		(* Check input high *)
		ELSIF
			BitInToCheck AND
			InputAvailable AND
			NOT CheckSignalLow AND
			CheckSignalHigh THEN

			TimerTimeOut(Start := FALSE, MTime := (sInit.MaxTime));
			State:=State_OK;
	
		(* Check signal high and input is low*)
		ELSIF
			NOT BitInToCheck AND
			InputAvailable AND
			NOT CheckSignalLow AND
			CheckSignalHigh THEN

			TimerTimeOut(Start := TRUE, MTime := (sInit.MaxTime));
			State:=STATE_ERROR (*INPUT_CHECKHIGH*);
			FB_ReadXmlLineMsg.ID:='SensorFaultNotHigh';

			TempErrorText:=sVisu.InstName;
			TempErrorText:=CONCAT(TempErrorText,' :');
			TempErrorText:=CONCAT(TempErrorText,sVisu.Description);
			TempErrorText:=CONCAT(TempErrorText,'  ');
			TempErrorText:=CONCAT(TempErrorText,FB_ReadXmlLineMsg.Text);

			Error.No:=2;
		ELSE
			TimerTimeOut(Start := FALSE, MTime := (sInit.MaxTime));

			IF	SetSignalHigh AND
				CheckSignalLow AND
				NOT PulseOn AND
				NOT FlashSignal AND
				NOT CheckSignalHigh AND
				NOT CheckSignalLow THEN

				State:=STATE_WAIT;
			END_IF
		END_IF

		(* Timeout check high *)
		IF	TimerTimeOut.Timeout AND
			NOT ResetIntern AND
			State=INPUT_CHECKHIGH 	THEN

			State:=STATE_ERROR (*INPUT_CHECKHIGHFAULT*);
			FB_ReadXmlLineMsg.ID:='NotHhigh';

			TempErrorText:=sVisu.InstName;
			TempErrorText:=CONCAT(TempErrorText,' ');
			TempErrorText:=CONCAT(TempErrorText,sVisu.Description);
			TempErrorText:=CONCAT(TempErrorText,' ');
			TempErrorText:=CONCAT(TempErrorText,FB_ReadXmlLineMsg.Text);
			Error.No:=3;
		END_IF
		(* Timeout check low *)
		IF	TimerTimeOut.Timeout AND
			NOT ResetIntern AND
			State=INPUT_CHECKLOW THEN

			State:=STATE_ERROR (*INPUT_CHECKLOWFAULT*);
			FB_ReadXmlLineMsg.ID:='NotLow';

			TempErrorText:=sVisu.InstName;
			TempErrorText:=CONCAT(TempErrorText,' ');
			TempErrorText:=CONCAT(TempErrorText,sVisu.Description);
			TempErrorText:=CONCAT(TempErrorText,' ');
			TempErrorText:=CONCAT(TempErrorText,FB_ReadXmlLineMsg.Text);
			Error.No:=4;
		END_IF

	ELSE	(* No action *)
		(* Reset ok signal*)
		IF 	State = State_OK AND
			StateOK_CycleFlag THEN

			State:=STATE_WAIT;
		END_IF
	END_IF

END_IF	(* Init ok *)

(*--------------------------------------------------------------------
	Updating processtime (if State_RUN, STATE_ERROR, STATE_RESETS, or STATE_STOPPED)
--------------------------------------------------------------------*)
IF	( State=State_RUN OR
	State=STATE_ERROR OR
	State=STATE_RESETS OR
	State=STATE_STOPPED ) AND
	sInit.MaxTime<>0 AND
	InputAvailable<>0 THEN

	TimerTimeOut;
	ProcessTime:=TimerTimeOut.PTime;
END_IF

(*------------------------------------------------------------------
	Reset-Handling
  ------------------------------------------------------------------*)
ResetIntern:=Reset;

IF 	ResetIntern THEN

	TimerTimeOut (Start := FALSE, MTime := (sInit.MaxTime));
	State:= STATE_RESETS;
	BitOutToSet:=FALSE;
	SetOutPulse(IN:=FALSE);
	TimerOn(IN:=FALSE);
	TimerOff(IN:=FALSE);

	SetSignalHigh:=FALSE;		 		 	(* Signal set  HIGH *)
	SetSignalLow:=FALSE;		 			(* Signal set  LOW  *)
	PulseOn:=FALSE;		 			(* Signal pulse On *)
	FlashSignal:=FALSE;		 			(* Signal FLASH  *)
ELSE  (* IF Reset=FALSE *)
	IF 	State=STATE_RESETS THEN
		State:=STATE_WAIT;
	END_IF
END_IF

(*------------------------------------------------------------------
	Clear all input variables
  ------------------------------------------------------------------*)
Reset:= FALSE;
SetSignalLow:=FALSE;
SetSignalHigh:=FALSE;
PulseOn:=FALSE;
FlashSignal:=FALSE;
CheckSignalLow:= FALSE;
CheckSignalHigh:= FALSE;

(*------------------------------------------------------------------
	HomePosition
  ------------------------------------------------------------------*)
HomePositionInfo:=State_OK;

(* Check input signal *)
IF	sInit.HomePosSignal=0 AND
	BitInToCheck AND
	InputAvailable THEN
	HomePositionInfo:=11;
END_IF

IF	sInit.HomePosSignal=1 AND
	NOT BitInToCheck AND
	InputAvailable THEN
	HomePositionInfo:=10;
END_IF

(* Check output signal *)
IF	sInit.HomePosOutput=0 AND
	BitOutToSet AND
	OutputAvailable THEN
	HomePositionInfo:=21;
END_IF

IF	sInit.HomePosOutput=1 AND
	NOT BitOutToSet AND
	OutputAvailable THEN
	HomePositionInfo:=20;
END_IF


(* Generating home position*)
(* Zuweisung der Grundstellung*)
IF HomePositionInfo=State_OK THEN
	HomePosition:= TRUE;
ELSE
	HomePosition:= FALSE;
	ListHomeNOK(InstName:=sInit.InstName,Description:=FB_ReadXmlLineConf.Text);
END_IF

(* Objekt-Grundstellung verknüpfen mit GesamtGrundstellung *)
(* object-homeposition concat with mainhomeposition *)
gHomeOk:=gHomeOk AND HomePosition;

(*------------------------------------------------------------------
	Set Visu-Vars
  ------------------------------------------------------------------*)
sVisu.BitInName			:= sInit.BitInName;
sVisu.BitOutToSet		:= BitOutToSet;
sVisu.BitInToCheck		:= BitInToCheck;
sVisu.State				:= State;
sVisu.HomePosition		:= HomePosition;


(*Copy output-signal to output-var*)
SignalOut:=BitOutToSet;
(*Copy input-signal to output-var*)
SignalIn:=BitInToCheck;

(*------------------------------------------------------------------
	Error-Handling
  ------------------------------------------------------------------*)
ErrorElapsed(CLK:= Error.Text<>'');
IF ErrorElapsed.Q THEN
	Error.DateTime:=gVarDTSystemtime;
END_IF

IF Error.Text<>''	AND ST_Lng.b_EndChangeLng THEN
	Error.Typ:=0;

	(*Error.DateTime:=;*)
	ErrorHandler.AddError(
			ErrorToAdd:=Error,
			sVisu:=Visu.ErrorHandler);
END_IF

IF 	NOT Enable AND ModeSelect.Mode=MODE_MANUAL AND
	Error.Text='' AND
	strAnlayse<>'' THEN

	strAnlayse:=CONCAT(' +++ gesperrt durch : ',strAnlayse);

	LaufschriftAnalyse(
	N:= 40,
	StepWidth:=1,
	PT:= t#100ms ,
	Text:= strAnlayse,
	Display=>sVisu.ErrorString );

	strAnlayse:='';
ELSE
	IF Error.Text<>''	THEN
		TempString:=CONCAT(' --- ',Error.Text);
		LaufschriftObj(
		N:= 40,
		StepWidth:=1,
		PT:= t#100ms ,
		Text:= TempString,
		Display=>sVisu.ErrorString );
	ELSE
		sVisu.ErrorString:='';
	END_IF
END_IF

sVisu.InstName:=sInit.InstName;
sVisu.BitOutName:=sInit.BitOutName;
sVisu.BitInName:=sInit.BitInName;
sVisu.ErrorPresent:=Error.Text<>'';

FB_ReadXmlLineConf(
	Prefix:= 'CONFIG',
	ID:= sInit.InstName,
	File:= 'CONFIG.xml',
	Text=> sVisu.Description);

FB_ReadXmlLineMsg(
	Prefix:= 'MSG',
	ID:= ,
	File:= 'MSG.xml',
	Text=>);

IF 	State = STATE_ERROR THEN
	TempErrorText:=sInit.BitInName;
	TempErrorText:=CONCAT(TempErrorText,' :');
	TempErrorText:=CONCAT(TempErrorText,sVisu.Description);
	TempErrorText:=CONCAT(TempErrorText,' -> ');
	TempErrorText:=CONCAT(TempErrorText,FB_ReadXmlLineMsg.Text);
END_IF
END_FUNCTION_BLOCK

(* POU zLibrary/AnaIn/FB_Encoder, ST *)
FUNCTION_BLOCK FB_Encoder
VAR_INPUT
	sInit					:sEncoderInit;	(* Initializingvalues to the Instance *)
	Reset					:BOOL;
END_VAR
VAR_OUTPUT
	State					:StateObject;	(* State of the object *)
	rpmValue			: LREAL;		(* rpm *)
	posValue			: LREAL;		(* mm *)
	Drehrichtung		: enum_Drehrichtung;
END_VAR
VAR_IN_OUT
	sVisu				:sEncoderVisu;
END_VAR
VAR

	Error					:ErrorStruct;
	TempErrorText			:STRING(255);
	ErrorElapsed			:BOOL;
	LaufschriftErrh			:FB_Laufschrift;
	LaufschriftObj			:FB_Laufschrift_STR255;
	InitState				:BOOL:=FALSE;	(* Internal State for initialising *)



	FB_ReadXmlLineConf		:FB_ReadXmlLine;
	FB_ReadXmlLineMsg		:FB_ReadXmlLine;
END_VAR


(*==================================================================*)
VAR_OUTPUT

END_VAR

VAR
	fb_ton_Reset		: TON;
	fb_ton_steht		: TON;
	fb_ton_dreht		: TON;

	fb_rTrigReset		: R_TRIG;
	fb_rTrigUnderflow		: R_TRIG;
	fb_rTrigOverflow		: R_TRIG;

	i_count_ueberlauf		: DINT;		(* +- 64bit *)
	lr_xBit		: LREAL;
	lr_rpmHelp	: LREAL;	(*°*)

	
	e_Value					AT %I* : UINT;		(* 65535 *)
	e_CountUnderflow		AT %I* : BOOL;
	e_CountOverflow			AT %I* : BOOL;
	a_CountReset			AT %Q* : BOOL;

END_VAR
VAR CONSTANT



END_VAR
Error.No:=0;
Error.Text:='';

(*------------------------------------------------------------------
	Initialization
  ------------------------------------------------------------------*)
IF  NOT InitState THEN
	InitState:=TRUE;
	State:=STATE_OK;
	(* Check instance name *)
	IF 	sInit.InstName=''THEN
		InitState:=FALSE;
		State:=STATE_ERROR;
		FB_ReadXmlLineMsg.ID:='InstNameNotDefined';

		TempErrorText:=sInit.BitInName;
		TempErrorText:=CONCAT(TempErrorText,' :');
		TempErrorText:=CONCAT(TempErrorText,sVisu.Description);
  		TempErrorText:=CONCAT(TempErrorText,' -> ');
		TempErrorText:=CONCAT(TempErrorText,FB_ReadXmlLineMsg.Text);
		Error.No:=4;
	(*CheckDescription*)
	ELSIF
		sInit.Description=''THEN
		InitState:=FALSE;
		State:=STATE_ERROR;
		FB_ReadXmlLineMsg.ID:='DescriptionNotDefined';

		TempErrorText:=sInit.BitInName;
		TempErrorText:=CONCAT(TempErrorText,' :');
		TempErrorText:=CONCAT(TempErrorText,sVisu.Description);
  		TempErrorText:=CONCAT(TempErrorText,' -> ');
		TempErrorText:=CONCAT(TempErrorText,FB_ReadXmlLineMsg.Text);
		Error.No:=4;
	ELSIF
		sInit.i_InkProRpm=0THEN
		InitState:=FALSE;
		State:=STATE_ERROR;
		FB_ReadXmlLineMsg.ID:='InkProRpmNotDefined';

		TempErrorText:=sInit.BitInName;
		TempErrorText:=CONCAT(TempErrorText,' :');
		TempErrorText:=CONCAT(TempErrorText,sVisu.Description);
  		TempErrorText:=CONCAT(TempErrorText,' -> ');
		TempErrorText:=CONCAT(TempErrorText,FB_ReadXmlLineMsg.Text);
		Error.No:=4;
	END_IF

END_IF

(* Add InitState to Global-Init-State to collect all Objects *)
gInitCollect:=gInitCollect AND InitState;

(*==================================================================*)
IF  InitState THEN
	(* Drehrichtung ermitteln *)
	fb_ton_steht(PT:=T#50MS);
	IF	lr_rpmHelp > rpmValue - 0.0001 AND
		lr_rpmHelp < rpmValue + 0.0001 THEN
		fb_ton_steht.IN:=TRUE;
		IF	fb_ton_steht.Q THEN
			Drehrichtung:= STEHT;
		END_IF
	ELSIF
		lr_rpmHelp < rpmValue THEN
		fb_ton_steht.IN:=FALSE;
		Drehrichtung:= VORWAERTS;
	ELSIF
		lr_rpmHelp > rpmValue THEN
		fb_ton_steht.IN:=FALSE;
		Drehrichtung:= RUECKWAERTS;
	END_IF
	lr_rpmHelp:=rpmValue;
	
	(* Encoderüberlauf*)
	fb_rTrigUnderflow(CLK:= e_CountUnderflow);
	fb_rTrigOverflow(CLK:= e_CountOverflow);
	IF 	fb_rTrigUnderflow.Q THEN
		i_count_ueberlauf:=i_count_ueberlauf - 1;
	ELSIF
		fb_rTrigOverflow.Q THEN
		i_count_ueberlauf:=i_count_ueberlauf + 1;
	END_IF

	(* bei Reset Nullen *)
	fb_ton_Reset(IN:=Reset , PT:= T#300MS , Q=> , ET=> );
	a_CountReset:=Reset OR sVisu.Reset;
	fb_rTrigReset(CLK:=fb_ton_Reset.Q, );
	IF	fb_rTrigReset.Q THEN
		Reset:=FALSE;
	END_IF

	(* aktuelle Position *)
	IF	e_Value <> 0 THEN
		lr_xBit:=EXPT(2,16);												(* 16 bit=65535  Inkremente Encoder*)
		rpmValue:= e_Value + (lr_xBit * DINT_TO_LREAL(i_count_ueberlauf));	(* Inkremente*)
		rpmValue:= rpmValue / sInit.i_InkProRpm;							(* Umdrehungen in Grad*)
	ELSE
		rpmValue:= 0;
		i_count_ueberlauf:=0;
	END_IF
	IF	sInit.lr_LaengeProRpm > 0 THEN
		posValue:= rpmValue * sInit.lr_LaengeProRpm;					(* Strecke in mm*)
	ELSE
		posValue:= 0;													(* Strecke in mm*)
	END_IF

	sVisu.posValue:=posValue;
	sVisu.rpmValue:=rpmValue;
	sVisu.Drehrichtung:=Drehrichtung;
END_IF
(* ------------------------------------------------------------------------------------------ *)
(* ---------------- LANGUAGE auslesen aus der XML Datei-------- *)
(* ------------------------------------------------------------------------------------------ *)
sVisu.BitInName:=sInit.BitInName;
sVisu.InstName:=sInit.InstName;
sVisu.ErrorPresent:=Error.Text<>'';

(*  *)
IF 	State=STATE_ERROR AND
	NOT ErrorElapsed THEN
	ErrorElapsed:=TRUE;
	Error.DateTime:=gVarDTSystemtime;
ELSIF
	State<>STATE_ERROR THEN
	ErrorElapsed:=FALSE;
	TempErrorText:='';
END_IF;

IF 	Error.Text<>'' AND
	ST_Lng.b_EndChangeLng THEN
	(*Error.DateTime:=;*)
	Error.Typ:=0;
	ErrorHandler.AddError(ErrorToAdd:=Error,
	sVisu:=Visu.ErrorHandler);
END_IF


FB_ReadXmlLineConf(
	Prefix:= 'CONFIG',
	ID:= sInit.InstName,
	File:= 'CONFIG.xml',
	Text=> sVisu.Description  );

FB_ReadXmlLineMsg(
	Prefix:= 'MSG',
	ID:= ,
	File:= 'MSG.xml',
	Text=>);

IF 	State = STATE_ERROR THEN
	TempErrorText:=sInit.BitInName;
	TempErrorText:=CONCAT(TempErrorText,' :');
	TempErrorText:=CONCAT(TempErrorText,sVisu.Description);
	TempErrorText:=CONCAT(TempErrorText,' -> ');
	TempErrorText:=CONCAT(TempErrorText,FB_ReadXmlLineMsg.Text);
END_IF


LaufschriftErrh(
N:= 160,
StepWidth:=1,
PT:= t#100ms ,
Text:= TempErrorText,
Display=>Error.Text );

LaufschriftObj(
N:= 40,
StepWidth:=1,
PT:= t#100ms ,
Text:= TempErrorText,
Display=>sVisu.ErrorString );
END_FUNCTION_BLOCK

(* POU zLibrary/EpsonRobot/FB_EpsonRobot, ST *)
FUNCTION_BLOCK FB_EpsonRobot (*25.NOV 2010, Bernd Happach*)
VAR_INPUT
	ExecuteMove					: BOOL; 				(* Move to PositionNo *)
	PosNo							: DINT;					(* Position No from Robot *)
	PosOffset						: DINT;					(* Offset *)
	Override						: DINT;					(* Global override *)
	OffsetX							: REAL;					(* Offset X *)
	OffsetY							: REAL;					(* Offset Y *)
	OffsetZ							: REAL;					(* Offset Z *)
	ApplPara						: ARRAY[0..7] OF	REAL; (* Machinespecific Values *)

	SetToolOn						: BOOL;
	SetToolOff						: BOOL;

	Vel								: DINT;					(* Velocity for Linear Movements *)
	Acc								: DINT;					(* Acceleration 0..100% *)

	Enable							: BOOL; 				(* Enables the operations on the valve *)
	Reset							: BOOL; 				(* switch for resetting the object *)
	SFCCurrentStep					: STRING(80);			(* aktually step in the step flow chart *)
	SFCCurrentPOU					: STRING(80);			(* Name of the step flow chart *)
	sInit								: sEpsonRobotInit;		(* Initializingvalues to the Instance *)
	sToolSettings					: sEpsonRobotToolSettings;
	strAnlayse						: STRING(255);  		(*String to analyse Lockings*)

	CollisionActivated			:BOOL;
	Tool2Unit_AST						:BOOL;
END_VAR
VAR_OUTPUT
	State							: StateObject;			(* State of the object *)
	HomePosition					: BOOL;					(* object in home-position*)
	ActualPosition					: DINT;
	ActualArea						: DINT;
END_VAR
VAR_IN_OUT
	sVisu							: sEpsonRobotVisu;   	(* Structure for Visualisation *)
END_VAR
VAR
	RemOutStart					AT %Q* :	BOOL; 		(* Startbit für Task Main *)
	RemOutStop					AT %Q* :	BOOL; 		(* Task stoppen/ beenden *)
	RemOutPause					AT %Q* :	BOOL; 		(* Task anhalten *)
	RemOutCont					AT %Q* :	BOOL; 		(* Task fortsetzen *)
	RemOutReset					AT %Q* :	BOOL; 		(* Reset auf Roboter *)
	RemOutPowerOn				AT %Q* :	BOOL; 		(* Armleistung ein *)
	RemOutPowerOff				AT %Q* :	BOOL; 		(* Armleistung aus *)
	RemOutPowerHi					AT %Q* :	BOOL; 		(* Motor hohe Leistung ein *)
	RemOutSetToolOn				AT %Q* :	BOOL; 		(* Anforderung Ausgang Robotertool EIN *)
	RemOutSetToolOff				AT %Q* :	BOOL; 		(* Anforderung Ausgang Robotertool AUS *)

	RemInReady					AT %I* :	BOOL; 		(* Betriebsbereit von Roboter *)
	RemInRunning					AT %I* :	BOOL; 		(* Task (Main) aktiv von Roboter *)
	RemInPaused					AT %I* :	BOOL; 		(* Task angehalten - nicht abgebrochen! *)
	RemInError						AT %I* :	BOOL; 		(* quittierbare Störung von Roboter *)
	RemInEStopOn					AT %I* :	BOOL; 		(* Notaus-Kreis aktiv von Roboter *)
	RemInSafeguardOn				AT %I* :	BOOL; 		(* Schutzkreis (Türen) aktiv von Roboter *)
	RemInSError					AT %I* :	BOOL; 		(* nicht quittierbare Störung - Roboter AEG notwendig *)
	RemInWarning					AT %I* :	BOOL; 		(* Warnmeldung von Roboter *)
	RemInTcpIP_Wait				AT %I* :	BOOL; 		(* Handshake TcpIp-Verbindung *)
	RemInAreaBit1					AT %I* :	BOOL; 		(* Bereichsüberwachung Bit 1 *)
	RemInAreaBit2					AT %I* :	BOOL; 		(* Bereichsüberwachung Bit 2 *)
	RemInAreaBit4					AT %I* :	BOOL; 		(* Bereichsüberwachung Bit 4 *)

	RemInToolCoilA					AT %I* :  BOOL;		(* Rückmeldung Tool CoilA/ Ausgang 1 ist ein *)
	RemInToolCoilB					AT %I* :  BOOL;		(* Rückmeldung Tool CoilB/ Ausgang 2 ist ein *)
	RemInToolInitSensor				AT %I* :  BOOL;		(* Tool Ruhesensor *)
	RemInToolWorkSensor			AT %I* :  BOOL;		(* Tool Ruhesensor *)

	CollisionSensor					AT %I* :  BOOL;		(* Kollisonssensor Greifer*)

(* Internal used variables for movement Handling *)
	WorkingStep				: DINT;					(* Index for StateMachine *)
	PosNoLastMove				: DINT;					(* Position No from Robot *)
(* Init Handling *)
	InitStep						: INT;					(* Init Step StateMachine *)
	InitState						: BOOL :=	FALSE;		(* Internal State for initialising *)
	InitTimeOut					: TON;

	StepTimeOut				: TON;
(* Tool Handling *)
	ManToolOn					: TP;
	ManToolOff					: TP;

(* Error Handling *)
	TP_RemOutReset			: TP;

	TimerTimeOut				: CheckProcTime;	(* Timer generates timeout signal *)
	ProcessTime				: DINT;				(* Counts the time since starting operation *)

	Error						: ErrorStruct;
	ErrorElapsed				: R_TRIG;

	LaufschriftErrh				:FB_Laufschrift_STR255;
	LaufschriftObj				:FB_Laufschrift_STR255;
	LaufschriftAnalyse			:FB_Laufschrift_STR255;
	TempString					:STRING(255);

(* Internal used Variables tp send/receife data over TcpIP Socket *)
	ConnectionAlive				: BOOL;
	ConnectionTimer			: TON;
	TcpIP_Wait					: TON;
	ToolTimeOut				: TON;

	FP_Connected				: R_TRIG;


	DataIn						: sEpsonRobotRecvData;
	DataOut					: sEpsonRobotSendData;
	DataOutOld					: sEpsonRobotSendData;
	SendString					: STRING(255);

	ReceiveStep				: INT;

	FBClientServerConnection	: FB_ClientServerConnection;
	FBSocketReceive			: FB_SocketReceive;
	FBSocketSend				: FB_SocketSend;
	SocketHandle				: T_HSOCKET;

	_TON_SEND				: TP;

	eSocketState 				: E_SocketConnectionState;
	rxBuffer						: STRING(255);
	recString					: STRING(255);
	recBytes					: UDINT;

	StringWork					: STRING(255);
	ItemNo						: INT;
	StringStart					: INT;
	StringEnd					: INT;
	StringLen					: INT;
	ItemString					: STRING(255);
	ItemStringArray				: ARRAY [1..20] OF STRING;
	iPosArray					: INT;
(* Constants *)
	Delim						: STRING	:= ',';
	NoOfItems					: INT 		:= 16;


(* Visu Handling *)
	BtnMove					: VisuButton;
	BtnReset					: VisuButton;
	BtnPrgStart					: VisuButton;
	BtnPrgStop					: VisuButton;

	BtnToolOn					: VisuButton;
	BtnToolOff					: VisuButton;


	FB_ReadXmlLineConf		: FB_ReadXmlLine;
	FB_ReadXmlLineMsg		: FB_ReadXmlLine;

(*Kollisionsüberwachung*)
	fb_ton_collision				:TON;
	b_collision							: BOOL;
END_VAR
VAR CONSTANT
	RecBufferLen				: DINT := 100;
END_VAR
ToolTimeOut(IN:=,PT:=DINT_TO_TIME(sInit.ToolMaxTime));
Error.No:=0;
Error.Text:='';

Collision();
(*------------------------------------------------------------------
	Initialization
  ------------------------------------------------------------------*)
InitTimeOut(In:=NOT InitState,Pt:=T#5s);
IF 	NOT InitState THEN
	CASE InitStep OF
		0: (* Init Instance *)
			InitStep:=10;

		10:	InitStep:=50;
	
		50: (*Check IP-adress and Port*)
			InitStep:=100;

		100: (* Init Done *)
			IF	sInit.InstName <> '' THEN

				FOR iPosArray:=1 TO 20 DO
					(*Übersetzungen stehen in der CONFIG.xml*)
					sVisu.PosArray[iPosArray]:= '';
					sVisu.PosArray[iPosArray]:= CONCAT(	sVisu.PosArray[iPosArray],	sInit.InstName);
					sVisu.PosArray[iPosArray]:= CONCAT(	sVisu.PosArray[iPosArray],	'.PosArray[');
					sVisu.PosArray[iPosArray]:= CONCAT(	sVisu.PosArray[iPosArray],	INT_TO_STRING(iPosArray));
					sVisu.PosArray[iPosArray]:= CONCAT(	sVisu.PosArray[iPosArray],	']');
				END_FOR

			InitState:=TRUE;
			END_IF
	END_CASE

END_IF

IF InitState THEN
(*------------------------------------------------------------------
	Show and Read Visu Buttons
  ------------------------------------------------------------------*)
	BtnMove(	Button:=sVisu.BtnMove,
				Enable:=ModeSelect.Mode =	MODE_MANUAL AND
											Enable AND
											State=STATE_WAIT,
				TextOn:='Start'
							);

	BtnReset(	Button:=sVisu.BtnReset,
				Enable:=ModeSelect.Mode=MODE_MANUAL OR State=STATE_ERROR,
				TextOn:='Reset',
							);
	BtnPrgStart(	Button:=sVisu.BtnPrgStart,
				Enable:=ModeSelect.Mode=MODE_MANUAL ,
				TextOn:='Verbinden',
							);
	BtnPrgStop(	Button:=sVisu.BtnPrgStop,
				Enable:=ModeSelect.Mode=MODE_MANUAL ,
				TextOn:='Trennen',
							);
	BtnToolOn(	Button:=sVisu.BtnToolOn,
				Enable:=ModeSelect.Mode=MODE_MANUAL AND RemInRunning AND State=STATE_WAIT,
				TextOn:=sToolSettings.NameBtnToolOn,
							);
	BtnToolOff(	Button:=sVisu.BtnToolOff,
				Enable:=ModeSelect.Mode=MODE_MANUAL AND RemInRunning AND State=STATE_WAIT,
				TextOn:=sToolSettings.NameBtnToolOff,
							);
(*------------------------------------------------------------------
	EA-Handling
  ------------------------------------------------------------------*)
	ActualArea.0:=RemInAreaBit1;
	ActualArea.1:=RemInAreaBit2;
	ActualArea.2:=RemInAreaBit4;

	sVisu.ActualArea:=ActualArea;
(*------------------------------------------------------------------
	Manual Mode
  ------------------------------------------------------------------*)
	IF 	ModeSelect.Mode=MODE_MANUAL AND
		Enable THEN
		ExecuteMove:= BtnMove.Pressed;
		Reset:=Reset OR BtnReset.Pressed;
		IF 	ExecuteMove THEN
			(*Override:=10;*)
			PosNo:=sVisu.PosNo;
			OffsetX:=sVisu.OffsetX;
			OffsetY:=sVisu.OffsetY;
			OffsetZ:=sVisu.OffsetZ;
		END_IF

		ManToolOn(In:=BtnToolOn.Pressed,Pt:=T#1s);
		ManToolOff(In:=BtnToolOff.Pressed,Pt:=T#1s);
	END_IF

	RemOutPowerHi:=ModeSelect.Mode>MODE_MANUAL;
(*------------------------------------------------------------------
	Move-Handling
  ------------------------------------------------------------------*)
	TP_RemOutReset(In:=Reset,PT:=T#1s);

	RemOutReset:=	TP_RemOutReset.Q AND
					(	(	RemInError AND ( DataIn.ErrorCode < 8000 OR DataIn.ErrorCode > 8999 )	) OR
						RemInEStopOn OR
						RemInWarning OR
						RemInSError OR
						RemInSafeguardOn OR
						RemInPaused
						);
	RemOutPowerOff:=TP_RemOutReset.Q;
	RemOutCont:=TP_RemOutReset.Q;

	RemOutStart := 	(RemInReady AND
					NOT RemInRunning AND
					NOT RemInError AND
					NOT RemInEStopOn AND
					NOT RemInSafeguardOn AND
					NOT RemInSError AND
					NOT RemInWarning AND
					NOT TP_RemOutReset.Q AND
					vGlbImpuls_0500ms AND
					ModeSelect.Mode>MODE_MANUAL
					)	OR
					(RemInReady AND
					NOT RemInRunning AND
					NOT RemInError AND
					NOT RemInEStopOn AND
					NOT RemInSafeguardOn AND
					NOT RemInSError AND
					NOT RemInWarning AND
					NOT TP_RemOutReset.Q AND
					ModeSelect.Mode=MODE_MANUAL AND
					BtnPrgStart.Pressed
					);

	RemOutStop:= 	RemInRunning AND
					ModeSelect.Mode=MODE_MANUAL AND
					(BtnPrgStop.Pressed OR TP_RemOutReset.Q) OR
					RemInRunning AND
					ModeSelect.Mode>MODE_MANUAL AND
					TP_RemOutReset.Q;

	RemOutSetToolOn:=	(    ManToolOn.Q AND ModeSelect.Mode=MODE_MANUAL ) OR
						(    SetToolOn  AND ModeSelect.Mode>MODE_MANUAL );

	RemOutSetToolOff:=	 (  ManToolOff.Q AND ModeSelect.Mode=MODE_MANUAL ) OR
						 (  SetToolOff AND ModeSelect.Mode>MODE_MANUAL );

(* Generate Flags To Start Movement *)

	CASE WorkingStep OF
	0: (* State STATE_WAIT *)

		State:=STATE_WAIT;

		IF 	ExecuteMove THEN
			WorkingStep:=10;
			(* Start Execution Time *)
			TimerTimeOut.Start:=TRUE;
			State:=STATE_RUN;
		END_IF
	10: (* Check Star Conditions *)
		IF  ConnectionAlive AND
			RemInRunning THEN
			WorkingStep:=100;
		ELSE
			State:=STATE_ERROR;
		END_IF
	100:(* Handle Robot EA´s if nessecary *)
			StepTimeOut(In:=FALSE);
			WorkingStep:=200;
	200:(* Start Movement - Assign Variables *)

			PosNoLastMove:=PosNo + PosOffset;

			DataOut.TelNo:=2;
			DataOut.PosNo:=PosNo + PosOffset;
			DataOut.Override:=Override;
			DataOut.OffsetX:=OffsetX;
			DataOut.OffsetY:=OffsetY;
			DataOut.OffsetZ:=OffsetZ;
			DataOut.ApplPara:=ApplPara;
			DataOut.Vel:=Vel;
			DataOut.Acc:=Acc;

			StepTimeOut(In:=DataIn.TelNo<>0 AND DataIn.TelNo<>DataOut.TelNo,Pt:=DINT_TO_TIME(sInit.MaxTime));
			IF 	DataIn.TelNo=DataOut.TelNo THEN
				WorkingStep:=201;
				ActualPosition:=0;

			ELSIF StepTimeOut.Q THEN
				(* Error *)
				State:=STATE_ERROR;
				FB_ReadXmlLineMsg.ID:='StartError';
				Error.No:=1;
				Error.Text:=sInit.InstName;
				Error.Text:=CONCAT(Error.Text,': ');
				Error.Text:=CONCAT(Error.Text,sInit.Description);
				Error.Text:=CONCAT(Error.Text,' - ');
				Error.Text:=CONCAT(Error.Text,FB_ReadXmlLineMsg.Text);
				WorkingStep:=999;
			END_IF

	201:(* Dummy step *)
			StepTimeOut(In:=FALSE);
			WorkingStep:=210;

	210:(* Wait Movement Done *)
			StepTimeOut(In:=DataIn.PosNo <>0 AND DataIn.PosNo<>DataOut.PosNo,Pt:=DINT_TO_TIME(sInit.MaxTime));
			IF 	DataIn.PosNo=DataOut.PosNo THEN
				DataOut.TelNo:=0;
				DataOut.PosNo:=0;
				ActualPosition:=DataIn.PosNo;
				WorkingStep:=220;
			ELSIF
				StepTimeOut.Q THEN
				(* Error *)
				State:=STATE_ERROR;
				FB_ReadXmlLineMsg.ID:='PosNoNotDefined';
				Error.No:=1;
				Error.Text:=sInit.InstName;
				Error.Text:=CONCAT(Error.Text,': ');
				Error.Text:=CONCAT(Error.Text,sInit.Description);
				Error.Text:=CONCAT(Error.Text,' - ');
				Error.Text:=CONCAT(Error.Text,FB_ReadXmlLineMsg.Text);
				WorkingStep:=999;
			END_IF
	220:(* Quit Telegramm Done *)
			IF 	DataIn.PosNo=0 AND DataIn.TelNo=0 THEN
				IF 	SetToolOn AND sInit.WithToolHandling THEN
					WorkingStep:=300;
				ELSIF
					SetToolOff AND sInit.WithToolHandling THEN
					WorkingStep:=400;
				ELSE
					WorkingStep:=1000;
				END_IF
			END_IF
	300: (* Check tool in workposition *)
			IF sToolSettings.NameWorkSensor<>'xxxx' THEN
				ToolTimeOut.IN:=TRUE;
				IF 	RemInToolWorkSensor THEN
					WorkingStep:=1000;
				ELSIF
					ToolTimeOut.Q THEN
					State:=STATE_ERROR;
					FB_ReadXmlLineMsg.ID:='TimeoutToolWork';
					Error.No:=1;
					Error.Text:=sInit.InstName;
					Error.Text:=CONCAT(Error.Text,': ');
					Error.Text:=CONCAT(Error.Text,sInit.Description);
					Error.Text:=CONCAT(Error.Text,' - ');
					Error.Text:=CONCAT(Error.Text,FB_ReadXmlLineMsg.Text);
				END_IF
			ELSE
				WorkingStep:=1000;
			END_IF

	400: (* Check tool in initposition *)
			IF 	sToolSettings.NameInitSensor<>'xxxx' THEN
				ToolTimeOut.IN:=TRUE;
				IF 	RemInToolInitSensor THEN
					WorkingStep:=1000;
				ELSIF
					ToolTimeOut.Q THEN
					State:=STATE_ERROR;
					FB_ReadXmlLineMsg.ID:='TimeoutToolInit';
					Error.No:=1;
					Error.Text:=sInit.InstName;
					Error.Text:=CONCAT(Error.Text,': ');
					Error.Text:=CONCAT(Error.Text,sInit.Description);
					Error.Text:=CONCAT(Error.Text,' - ');
					Error.Text:=CONCAT(Error.Text,FB_ReadXmlLineMsg.Text);	
				END_IF
			ELSE
				WorkingStep:=1000;
			END_IF

	999: (* State Error *)
			State:=STATE_ERROR;
			StepTimeOut(In:=FALSE);
			TimerTimeOut.Start:=FALSE;
	1000: (* State OK *)
			State:=STATE_OK;
			TimerTimeOut.Start:=FALSE;
			ToolTimeOut.IN:=FALSE;
			IF 	NOT ExecuteMove THEN (*OR PosNoLastMove<>PosNo*)
				WorkingStep:=0;
				State:=STATE_WAIT;
				ProcessTime:=TimerTimeOut.PTime;
			END_IF
	END_CASE

(*--------------------------------------------------------------------
		Handle Timeout
  --------------------------------------------------------------------*)
	IF 	TimerTimeOut.Timeout AND
		State<>STATE_ERROR THEN

		State:=STATE_TIMEOUT;
		Error.No:=1;
		Error.Text:=sInit.InstName;
		Error.Text:=CONCAT(Error.Text,': ');
		Error.Text:=CONCAT(Error.Text,sInit.Description);
		Error.Text:=CONCAT(Error.Text,' - ');
		Error.Text:=CONCAT(Error.Text,' [Rob. Error code: ');
		Error.Text:=CONCAT(Error.Text,DINT_TO_STRING(DataIn.ErrorCode));
		Error.Text:=CONCAT(Error.Text,']');

		FB_ReadXmlLineMsg.ID:=DINT_TO_STRING(DataIn.ErrorCode);

		CASE DataIn.ErrorCode OF
			8000:
				Error.Text:=CONCAT(Error.Text,FB_ReadXmlLineMsg.Text);
			8001:
				Error.Text:=CONCAT(Error.Text,FB_ReadXmlLineMsg.Text);
			8002:
				Error.Text:=CONCAT(Error.Text,FB_ReadXmlLineMsg.Text);
			8003:
				Error.Text:=CONCAT(Error.Text,FB_ReadXmlLineMsg.Text);
			8006:
				Error.Text:=CONCAT(Error.Text,FB_ReadXmlLineMsg.Text);
			8010:
				Error.Text:=CONCAT(Error.Text,FB_ReadXmlLineMsg.Text);
			8011:
				Error.Text:=CONCAT(Error.Text,FB_ReadXmlLineMsg.Text);
			8012:
				Error.Text:=CONCAT(Error.Text,FB_ReadXmlLineMsg.Text);
			8013:
				Error.Text:=CONCAT(Error.Text,FB_ReadXmlLineMsg.Text);
			8014:
				Error.Text:=CONCAT(Error.Text,FB_ReadXmlLineMsg.Text);
			8015:
				Error.Text:=CONCAT(Error.Text,FB_ReadXmlLineMsg.Text);
			8016:
				Error.Text:=CONCAT(Error.Text,FB_ReadXmlLineMsg.Text);
		END_CASE
	END_IF

(*--------------------------------------------------------------------
		Call Timers
  --------------------------------------------------------------------*)
	TimerTimeOut(MTime:=sInit.MaxTime);

(*--------------------------------------------------------------------
		Updating processtime (if State_RUN, STATE_TIMEOUT, STATE_RESETS, or STATE_STOPPED)
  --------------------------------------------------------------------*)
	IF	(State=STATE_OK OR
		State=STATE_TIMEOUT OR
		State=STATE_RESETS OR
		State=STATE_STOPPED) AND
		 sInit.MaxTime<>0 THEN
		ProcessTime:=TimerTimeOut.PTime;
	END_IF

(*--------------------------------------------------------------------
	HomePosition
  --------------------------------------------------------------------*)
	IF 	(ActualPosition MOD 1000)=1 AND ConnectionAlive THEN
		HomePosition:=TRUE;
	ELSE
		HomePosition:=FALSE;
	END_IF

	(* Generating home position*)
	IF NOT HomePosition THEN
		ListHomeNOK(InstName:=sInit.InstName,Description:=FB_ReadXmlLineConf.Text);
	END_IF

	(* Object-homeposition concat with mainhomeposition *)
	gHomeOk:=gHomeOk AND HomePosition;

(*------------------------------------------------------------------
	Update Visu
  ------------------------------------------------------------------*)
	sVisu.InstName:=sInit.InstName;
	sVisu.Description:=sInit.Description;
	sVisu.TcpIpAdress:=sInit.TcpIPAdress;
	CASE eSocketState OF
		eSOCKET_CONNECTED: sVisu.SocketState:='Connected';
		eSOCKET_DISCONNECTED: sVisu.SocketState:='Disconnected';
		eSOCKET_SUSPENDED: sVisu.SocketState:='Suspended';
	END_CASE
	sVisu.State:=State;

	sVisu.ProcessTime:=ProcessTime;
	sVisu.HomePosition:=HomePosition;
	sVisu.ActualPosition:=ActualPosition;
	sVisu.ConnectionAlive:=ConnectionAlive;

	sVisu.PosX:=DataIn.PosX;
	sVisu.PosY:=DataIn.PosY;
	sVisu.PosZ:=DataIn.PosZ;

	sVisu.PosOffset:= 			PosOffset;

(* EA's from Robot *)
	sVisu.RemOutStart:=			RemOutStart; 		(* For Moving to WorkPosition *)
	sVisu.RemOutStop:=			RemOutStop; 		(* For Moving to WorkPosition *)
	sVisu.RemOutPause	:= 		RemOutPause; 		(* For Moving to WorkPosition *)
	sVisu.RemOutCont:=			RemOutCont; 		(* For Moving to WorkPosition *)
	sVisu.RemOutReset:=		RemOutReset; 		(* For Moving to WorkPosition *)
	sVisu.RemOutPowerOn:=	RemOutPowerOn; 		(* For Moving to WorkPosition *)
	sVisu.RemOutPowerOff:=	RemOutPowerOff; 		(* For Moving to WorkPosition *)
	sVisu.RemOutPowerHi:=		RemOutPowerHi; 		(* For Moving to WorkPosition *)

	sVisu.RemInReady:=			RemInReady; 		(* For Moving to WorkPosition *)
	sVisu.RemInRunning	:=		RemInRunning; 		(* For Moving to WorkPosition *)
	sVisu.RemInPaused:=		RemInPaused; 		(* For Moving to WorkPosition *)
	sVisu.RemInError:=			RemInError; 		(* For Moving to WorkPosition *)
	sVisu.RemInEStopOn:=		RemInEStopOn; 		(* For Moving to WorkPosition *)
	sVisu.RemInSafeguardOn:=	RemInSafeguardOn; 		(* For Moving to WorkPosition *)
	sVisu.RemInSError:=			RemInSError; 		(* For Moving to WorkPosition *)
	sVisu.RemInWarning	:=		RemInWarning; 		(* For Moving to WorkPosition *)

	sVisu.RemInTcpIP_Wait	:=	RemInTcpIP_Wait; 		(* For Moving to WorkPosition *)
	sVisu.RemInAreaBit1	:=		RemInAreaBit1; 		(* For Moving to WorkPosition *)
	sVisu.RemInAreaBit2	:=		RemInAreaBit2; 		(* For Moving to WorkPosition *)
	sVisu.RemInAreaBit4	:=		RemInAreaBit4; 		(* For Moving to WorkPosition *)

	sVisu.WithToolHandling:=		sInit.WithToolHandling;
	sVisu.NameCoilA:=				sToolSettings.NameCoilA;
	sVisu.NameCoilB:=				sToolSettings.NameCoilB;
	sVisu.NameInitSensor:=			sToolSettings.NameInitSensor;
	sVisu.NameWorkSensor:=		sToolSettings.NameWorkSensor;
	sVisu.RemInToolCoilA:=			RemInToolCoilA;
	sVisu.RemInToolCoilB:=			RemInToolCoilB;
	sVisu.RemInToolInitSensor:=		RemInToolInitSensor;
	sVisu.RemInToolWorkSensor	:=	RemInToolWorkSensor;
	sVisu.RemOutSetToolOn	:=		RemOutSetToolOn;
	sVisu.RemOutSetToolOff	:=		RemOutSetToolOff;

(*------------------------------------------------------------------
	Check ConnectionState
  ------------------------------------------------------------------*)
(* Toggle Alive Bit *)

	ConnectionTimer(IN:=DataOut.Alive<>DataIn.Alive OR eSocketState<>eSOCKET_CONNECTED , PT:= t#2000ms );
	ConnectionAlive:=NOT ConnectionTimer.Q;
	
	IF 	DataOut.Alive=DataIn.Alive OR
		(NOT ConnectionAlive AND eSocketState=eSOCKET_CONNECTED AND vGlbImpuls_1000ms) THEN
		IF DataOut.Alive=0 THEN
			DataOut.Alive:=1;
		ELSE
			DataOut.Alive:=0;
		END_IF
	END_IF

	IF 	eSocketState<>eSOCKET_CONNECTED THEN
		DataOut.Alive:=0;
	END_IF
(* Create Sendstring *)


	sendString:=CONCAT(DINT_TO_STRING(DataOut.Alive),Delim);
	sendString:=CONCAT(sendString,DINT_TO_STRING(DataOut.TelNo));
	sendString:=CONCAT(sendString,Delim);
	sendString:=CONCAT(sendString,DINT_TO_STRING(DataOut.PosNo));
	sendString:=CONCAT(sendString,Delim);
	sendString:=CONCAT(sendString,DINT_TO_STRING(DataOut.Override));
	sendString:=CONCAT(sendString,Delim);
	sendString:=CONCAT(sendString,DINT_TO_STRING(DataOut.Vel));
	sendString:=CONCAT(sendString,Delim);
	sendString:=CONCAT(sendString,DINT_TO_STRING(DataOut.Acc));
	sendString:=CONCAT(sendString,Delim);
	sendString:=CONCAT(sendString,REAL_TO_STRING(DataOut.OffsetX * 1000.0));
	sendString:=CONCAT(sendString,Delim);
	sendString:=CONCAT(sendString,REAL_TO_STRING(DataOut.OffsetY * 1000.0));
	sendString:=CONCAT(sendString,Delim);
	sendString:=CONCAT(sendString,REAL_TO_STRING(DataOut.OffsetZ * 1000.0));
	sendString:=CONCAT(sendString,Delim);
	sendString:=CONCAT(sendString,REAL_TO_STRING(DataOut.ApplPara[0] * 1000.0));
	sendString:=CONCAT(sendString,Delim);
	sendString:=CONCAT(sendString,REAL_TO_STRING(DataOut.ApplPara[1] * 1000.0));
	sendString:=CONCAT(sendString,Delim);
	sendString:=CONCAT(sendString,REAL_TO_STRING(DataOut.ApplPara[2] * 1000.0));
	sendString:=CONCAT(sendString,Delim);
	sendString:=CONCAT(sendString,REAL_TO_STRING(DataOut.ApplPara[3] * 1000.0));
	sendString:=CONCAT(sendString,Delim);
	sendString:=CONCAT(sendString,REAL_TO_STRING(DataOut.ApplPara[4] * 1000.0));
	sendString:=CONCAT(sendString,Delim);
	sendString:=CONCAT(sendString,REAL_TO_STRING(DataOut.ApplPara[5] * 1000.0));
	sendString:=CONCAT(sendString,Delim);
	sendString:=CONCAT(sendString,REAL_TO_STRING(DataOut.ApplPara[6] * 1000.0));
	sendString:=CONCAT(sendString,Delim);
	sendString:=CONCAT(sendString,REAL_TO_STRING(DataOut.ApplPara[7] * 1000.0));
	sendString:=CONCAT(sendString,Delim);

	FP_Connected(CLK:= eSocketState=eSOCKET_CONNECTED);

	IF 	(MEMCMP(ADR(DataOut),ADR(DataOutOld),SIZEOF(DataOut))<>0 AND eSocketState=eSOCKET_CONNECTED) OR FP_Connected.Q THEN
		FBSocketSend.bExecute:=TRUE;
		DataOutOld:=DataOut;
	END_IF

	TcpIP_Wait(IN:=RemInTcpIP_Wait , PT:=t#5ms );

	CASE ReceiveStep OF
	0: (* Waiting for Robot is Ready to Connect *)
		IF 	TcpIP_Wait.Q THEN
			ReceiveStep:=1;
		END_IF
	1: (* Connect *)
		FBClientServerConnection.bEnable:= TRUE;
		IF 	FBClientServerConnection.bBusy THEN
			ReceiveStep:=2;
		END_IF
	2:(* Connected *)
		IF 	eSocketState=eSOCKET_CONNECTED THEN
			ReceiveStep:=10;
		END_IF
	10:
		IF 	SocketHandle.handle>0 THEN
			ReceiveStep:=11;
		END_IF
	11:(* Start to Receive *)
		rxBuffer:='';
	 	FBSocketReceive.bExecute:=TRUE;
		IF 	FBSocketReceive.bBusy THEN
			ReceiveStep:=12;
		END_IF
	12:(* Rec Done *)
		FBSocketReceive.bExecute:=TRUE;
		IF 	NOT FBSocketReceive.bBusy AND NOT
			FBSocketReceive.bError AND
			FBSocketReceive.nRecBytes>99 THEN
			(* Data Received *)
			ReceiveStep:=20;
		ELSIF
			NOT FBSocketReceive.bBusy AND NOT
			FBSocketReceive.bError AND
			FBSocketReceive.nRecBytes=0 THEN
			(* NO Data Received *)
			ReceiveStep:=10;
		ELSIF
			NOT FBSocketReceive.bBusy AND NOT
			FBSocketReceive.bError AND
			FBSocketReceive.nRecBytes>0 THEN
			(* NO Data Received *)
			ReceiveStep:=10;

		ELSIF
			NOT FBSocketReceive.bBusy AND
			FBSocketReceive.bError THEN
			(* ERROR *)
			ReceiveStep:=100;
		END_IF
	20:(* Decrypt Data *)
		recString:=rxBuffer;
	  (* Handle String *)
		StringWork:=recString;
		FOR ItemNo:=1 TO NoOfItems DO
			StringStart:=1;
			StringEnd:=FIND(StringWork, Delim);
			IF 	StringEnd<>0 THEN
				StringLen:=StringEnd-StringStart;
				ItemString:=MID(StringWork,StringLen,StringStart);
				StringWork:=REPLACE(StringWork,'',StringLen+1,StringStart);
				ItemStringArray[ItemNo]:=ItemString;
			ELSE
				(* Delete $r and $n *)
				IF 	StringWork<>'' THEN
					StringStart:=FIND(StringWork, '$R');
					IF 	StringStart <> 0 THEN
						StringLen:=LEN(StringWork)-(StringStart-1);
						StringWork:=REPLACE(StringWork,'',StringLen,StringStart);
					END_IF

					StringStart:=FIND(StringWork, 'X');
					IF 	StringStart <> 0 THEN
						StringLen:=LEN(StringWork)-(StringStart-1);
						StringWork:=REPLACE(StringWork,'',StringLen,StringStart);
					END_IF

					StringStart:=FIND(StringWork, '$N');
					IF 	StringStart <> 0 THEN
						StringLen:=LEN(StringWork)-(StringStart-1);
						StringWork:=REPLACE(StringWork,'',StringLen,StringStart);
					END_IF

					ItemStringArray[ItemNo]:=StringWork;
				END_IF
				EXIT;
			END_IF
		END_FOR (* ItemNo *)

		ReceiveStep:=22;
	22: (*Check Data*)
		IF 	ItemStringArray[1]='BEG' THEN
			DataIn.Alive:=STRING_TO_DINT(ItemStringArray[2]);
			DataIn.TelNo:=STRING_TO_DINT(ItemStringArray[3]);
			DataIn.PosNo:=STRING_TO_DINT(ItemStringArray[4]);
			DataIn.PosX:=STRING_TO_REAL(ItemStringArray[5]) / 1000.0;
			DataIn.PosY:=STRING_TO_REAL(ItemStringArray[6]) / 1000.0;
			DataIn.PosZ:=STRING_TO_REAL(ItemStringArray[7]) / 1000.0;

			DataIn.ApplPara[0]:=STRING_TO_REAL(ItemStringArray[8]) / 1000.0;
			DataIn.ApplPara[1]:=STRING_TO_REAL(ItemStringArray[9]) / 1000.0;
			DataIn.ApplPara[2]:=STRING_TO_REAL(ItemStringArray[10]) / 1000.0;
			DataIn.ApplPara[3]:=STRING_TO_REAL(ItemStringArray[11]) / 1000.0;
			DataIn.ApplPara[4]:=STRING_TO_REAL(ItemStringArray[12]) / 1000.0;
			DataIn.ApplPara[5]:=STRING_TO_REAL(ItemStringArray[13]) / 1000.0;
			DataIn.ApplPara[6]:=STRING_TO_REAL(ItemStringArray[14]) / 1000.0;
			DataIn.ApplPara[7]:=STRING_TO_REAL(ItemStringArray[15]) / 1000.0;
			DataIn.ErrorCode	:=STRING_TO_DINT(ItemStringArray[16]);
			ReceiveStep:=10;
		ELSE
			ReceiveStep:=10;
		END_IF
	100: (* Errorhandler -> Reconnect *)
		FBClientServerConnection.bEnable:= FALSE;
		ReceiveStep:=101;

	101:
		IF	eSocketState=eSOCKET_DISCONNECTED THEN
			ReceiveStep:=0;
		END_IF
	END_CASE

	FBClientServerConnection(
		sSrvNetID:=	'',
		nMode:= CONNECT_MODE_ENABLEDBG,
		sRemoteHost:= sInit.TcpIPAdress,
		nRemotePort:= sInit.TcpIPSocket,
		tReconnect:= t#10s,
		hSocket=> SocketHandle,
		eState=> eSocketState);


	FBSocketReceive(
		sSrvNetId:= '',
		hSocket:= SocketHandle,
		cbLen:= RecBufferLen,
		pDest:= ADR(rxBuffer),
		tTimeout:= t#1s,
		nRecBytes=> recBytes);

	FBSocketReceive.bExecute:=FALSE;
	_TON_SEND(IN:=FBSocketSend.bExecute , PT:=t#10ms );
	FBSocketSend(
		sSrvNetId:= '',
		hSocket:= SocketHandle,
		cbLen:= LEN(sendString),
		pSrc:= ADR(sendString),
		tTimeout:= t#1s
	 );

	FBSocketSend.bExecute:=FALSE;

END_IF (* Init OK *)

(*------------------------------------------------------------------
	Reset-Handling
  ------------------------------------------------------------------*)
IF 	Reset THEN
	RemOutStart:=FALSE;
	RemOutStop:=TRUE;
	RemOutReset:=TRUE;
	State:=STATE_RESETS;
	WorkingStep:=0;
	ProcessTime:=0;
	TimerTimeOut.Start:=FALSE;
	DataOut.TelNo:=0;
	DataOut.PosNo:=0;
	DataOut.Alive:=0;
	b_collision:=FALSE;
	IF	NOT ConnectionAlive THEN
		ReceiveStep:=100;
	END_IF
END_IF


(*------------------------------------------------------------------
	Error-Handling
  ------------------------------------------------------------------*)
ErrorElapsed(CLK:= Error.Text<>'');
IF 	ErrorElapsed.Q THEN
	Error.DateTime:=gVarDTSystemtime;
END_IF

IF 	Error.Text<>'' AND
	ST_Lng.b_EndChangeLng THEN
	Error.Typ:=0;

	(*Error.DateTime:=;*)
	ErrorHandler.AddError(	ErrorToAdd:=Error,
							sVisu:=Visu.ErrorHandler);

END_IF

IF 	NOT Enable AND
	ModeSelect.Mode=MODE_MANUAL AND
	Error.Text='' AND
	strAnlayse<>'' THEN

	strAnlayse:=CONCAT(' +++ gesperrt durch : ',strAnlayse);

	LaufschriftAnalyse(
	N:= 40,
	StepWidth:=1,
	PT:= t#100ms ,
	Text:= strAnlayse,
	Display=>sVisu.ErrorString );

	strAnlayse:='';
ELSE
	IF 	Error.Text<>'' THEN
		TempString:=CONCAT(' --- ',Error.Text);
		LaufschriftObj(
		N:= 80,
		StepWidth:=1,
		PT:= t#100ms ,
		Text:= TempString,
		Display=>sVisu.ErrorString );
	ELSE
		sVisu.ErrorString:='';
	END_IF
END_IF
sVisu.ErrorPresent:=sVisu.ErrorString='';
(*------------------------------------------------------------------
	Reset Inputs
  ------------------------------------------------------------------*)

IF 	state=STATE_WAIT OR
	state=STATE_RESETS OR
	state=STATE_OK THEN
	ExecuteMove:=FALSE;
	PosNo:=0;
	Enable:=FALSE;
	Reset:= FALSE;
	SetToolOn:= FALSE;
	SetToolOff:= FALSE;

	(*Override:=	0;			(* Global override *)*)
	OffsetX	:=	0.0;			(* Offset X *)
	OffsetY	:=	0.0;			(* Offset Y *)
	OffsetZ	:=	0.0;			(* Offset Z *)
	ApplPara[0]:=0.0; 		(* Machinespecific Values *)
	ApplPara[1]:=0.0; 		(* Machinespecific Values *)
	ApplPara[2]:=0.0; 		(* Machinespecific Values *)
	ApplPara[3]:=0.0; 		(* Machinespecific Values *)
	ApplPara[4]:=0.0; 		(* Machinespecific Values *)
	ApplPara[5]:=0.0; 		(* Machinespecific Values *)
	ApplPara[6]:=0.0; 		(* Machinespecific Values *)
	ApplPara[7]:=0.0; 		(* Machinespecific Values *)

END_IF


sVisu.BitName:=sInit.BitName;
sVisu.InstName:=sInit.InstName;

FB_ReadXmlLineConf(
	Prefix:= 'CONFIG',
	ID:= sInit.InstName,
	File:= 'CONFIG.xml',
	Text=> sVisu.Description );

FB_ReadXmlLineMsg(
	Prefix:= 'MSG',
	ID:= ,
	File:= 'MSG.xml',
	Text=>);
END_FUNCTION_BLOCK
ACTION Collision:
fb_ton_collision(IN:=collisionSensor AND Tool2Unit_AST AND ActualArea = 6,PT:= t#100ms, Q=> , ET=> );
IF 	fb_ton_collision.Q THEN
	b_collision:= TRUE;
END_IF

IF CollisionActivated THEN
	IF 	b_collision THEN
		RemOutStart:=FALSE;
		RemOutStop:=TRUE;
		WorkingStep:=0;
		State:=STATE_ERROR;
		Error.Text:=CONCAT('Error movement: ','collision');
		Error.No:=1;
	END_IF
END_IF
END_ACTION

(* POU zLibrary/ept/BDE/Fb_ExportHydraString, ST *)
FUNCTION_BLOCK Fb_ExportHydraString
VAR_INPUT
	s_Path				: T_MaxString;
	s_system_time		: STRING;
	st_data				: struct_Hydra8;
	bKopiereDateiAufServer	: BOOL := FALSE;
	sDateiName			: STRING := 'Eingang.txt';
	tStartTime			: TIME := T#10S;
	sToolPath			: STRING(255) := '';
END_VAR
VAR
	fb_state_entry			: ST_StateEntry;
	fbFindFiles			: FB_EnumFindFileList;
	fbFindFilesEntry		: ST_FindFileEntry;
	fbFileOpen			: FB_FileOpen;
	fbFilePuts			: FB_FilePuts;
	fbFileClose			: FB_FileClose;
	HelpString			: T_MaxString;
	Substring			:ARRAY[1..3] OF STRING(255);
	fb_ton_start			: TON;
	hFile					:UINT;
	nErrIdOpen					:UDINT;
	nErrIdWrite					:UDINT;
	nErrIdClose					:UDINT;
	nErrIdCloseCounter			:UDINT;
	sFileName				:STRING;
	i						:UINT;

	i_dint_to_hydra		: DINT;
	s_dint_to_hydra	: STRING;

	sDatum		: STRING(10) := '01/01/1970';	(* aktuelles Datum im Format TT/MM/JJJJ *)
	sZeit		: STRING(8) := '00:00:00';	(* aktuelle Zeit im Format HH:MM:SS *)

	sPathStrDateiAufServerSpeichern	:T_MaxString;	(* Pfad damit Leerzeichen im Pfad erlaubt sind*)
	DateiAufServerSpeichern 		:NT_StartProcess;
END_VAR
VAR_OUTPUT
	Ready						:BOOL;
	Busy						:BOOL;
	Done						:BOOL;
	Error						:BOOL;
END_VAR
VAR CONSTANT
	sMSTAT					: STRING := 'MSTAT=';
	sDatumPrefix				: STRING := 'DAT=';
	sZeitPrefix				: STRING := 'ZEI=';
	sCounter					: STRING := 'COUNTER';
	sTrennzeichen			: STRING := '|';
	sDosGeraetePfad			: STRING(4) := '\\.\';	(* https://docs.microsoft.com/de-de/dotnet/standard/io/file-path-formats
	Das Windows-Betriebssystem verfügt über ein einheitliches Objektmodell,
	das auf alle Ressourcen, einschließlich Dateien, verweist. Sie können über
	das Konsolenfenster auf diese Objektpfade zugreifen. Diese werden über einen
	speziellen Ordner aus symbolischen Verknüpfungen, denen ältere DOS- und UNC-Pfade
	zugeordnet sind, für die Win32-Schicht zur Verfügung gestellt. Der Zugriff auf
	diesen speziellen Ordner erfolgt über die DOS-Gerätepfadsyntax, die einer der Folgenden entspricht:*)
END_VAR
(*======================================================
   FB: Fb_ExportHydraString
 ------------------------------------------------------
   Auth: 	Thomas Vilgis    						 
   Date: 	27.01.2022    						     
   Rev.: 		1.1	
   Desc:		Dieser Baustein übernimmt die Kommunikation zum neuen Hydra 8.
			Es wird alle 2 Sekunden (Zeit einstellbar) eine Textdatei mit den Produktionsdaten für
			das Hydra erstellt. Hydra liest diese Datei aus und löscht sie dann.
			Alle Daten werden in eine Zeile geschrieben
			Es gibt insgesamt 20 Zähler. Es werden aber nur die jeweils 4 letzten Ziffern übergeben.
			Fehlende Ziffern werden mit 0 aufgefüllt.
			Dann gibt es noch 999 Status-Bits. Das erste TRUE-Bit im  Array wird als Status übergeben.
			Außerdem werden noch die aktuelle Uhrzeit und das Datum übergeben.
			Auf Wunsch von Stanzerei Augsburg wurde aus diesem Baustein ein Fb gemacht.
			Per Vbs-Stript wird eine Batch-Datei gestartet, die die erzeugte txt-Datei auf den
			Server verschiebt. Dort soll eine zusätzliche Auswertung durchgeführt werden.
			NEU: Neuaufbau FB, da Filehandle zu Fehlern führt (D.Peichl 16.02.2022)
   Historie: 	1.1

 ========================================================*)



(* Zeiten *)
fb_ton_start(IN:= NOT fb_ton_start.Q, PT:= tStartTime, Q=>  , ET=> );


(* ======================================Schrittkette======================================== *)
fb_state_entry(i16_pos:= 1);

CASE fb_state_entry.i16_step OF
(*=======================================================*)
	INIT_OBJ: fb_state_entry.s_debugtext:='initialisieren';	

		(*-----------------------Weiterschaltbedingungen----------------------------*)
		IF fb_state_entry.fb_ton_Step.ET >= T#5S THEN
			fb_state_entry.i16_next_step:=BEREIT;
		END_IF

		IF fb_state_entry.X THEN
			sFileName:=CONCAT(s_Path,sDateiName);
			sPathStrDateiAufServerSpeichern := CONCAT(sDosGeraetePfad, sToolPath);
		END_IF

(*=======================================================*)
	BEREIT: fb_state_entry.s_debugtext:='Start';

		IF fb_state_entry.E THEN
			Ready := TRUE;
		END_IF

		(*-----------------------Weiterschaltbedingungen----------------------------*)
		IF fb_ton_start.Q THEN
			Error := FALSE;
			Busy := TRUE;
			Ready := FALSE;
			Done := FALSE;
			fb_state_entry.i16_next_step:=110;
		END_IF

(*=======================================================*)
	110: fb_state_entry.s_debugtext:='Prüfe, ob Datei geschlossen ist';

		(*-----------------------Weiterschaltbedingungen----------------------------*)
		IF hFile = 0 THEN
			fb_state_entry.i16_next_step:=120;
		ELSE
			fb_state_entry.i16_next_step:=112;
		END_IF
		
(*=======================================================*)
	112: fb_state_entry.s_debugtext:='Datei schließen';

		IF fb_state_entry.E THEN
			fbFileClose.bExecute:=TRUE;
		END_IF

		(*-----------------------Weiterschaltbedingungen----------------------------*)
		IF 	fbFileClose.bBusy THEN
			fb_state_entry.i16_next_step:=114;
		END_IF

(*=======================================================*)
	114: fb_state_entry.s_debugtext:='Datei schließen';

		(*-----------------------Weiterschaltbedingungen----------------------------*)
		IF NOT fbFileClose.bBusy THEN
			hFile := 0;
			fbFileClose.bExecute:=FALSE;
			IF 	fbFileClose.bError THEN
				nErrIdClose:=fbFileClose.nErrId;
				nErrIdCloseCounter := nErrIdCloseCounter + 1;
				fb_state_entry.i16_next_step:=FEHLER;
			ELSE
				fb_state_entry.i16_next_step:=120;
			END_IF
		END_IF

(*=======================================================*)
	120: fb_state_entry.s_debugtext:='Prüfe, ob Datei vorhanden ist';

		IF fb_state_entry.E THEN
			fbFindFiles.bExecute := TRUE;
		END_IF

		(*-----------------------Weiterschaltbedingungen----------------------------*)
		IF fbFindFiles.bBusy THEN
			fb_state_entry.i16_next_step:=130;
		END_IF

(*=======================================================*)
	130: fb_state_entry.s_debugtext:='Prüfe, ob Datei vorhanden ist';

		(*-----------------------Weiterschaltbedingungen----------------------------*)
		IF NOT fbFindFiles.bBusy THEN
			fbFindFiles.bExecute := FALSE;
			IF NOT fbFindFiles.bError THEN
				IF fbFindFiles.nFindFiles = 0 THEN
					fb_state_entry.i16_next_step:=140;
				ELSE
					fb_state_entry.i16_next_step:=300;	(* Datei noch vorhanden >> tue nichts *)
				END_IF
			ELSE
				fb_state_entry.i16_next_step:=FEHLER;
			END_IF
		END_IF
		
(*=======================================================*)
	140: fb_state_entry.s_debugtext:='Counter 1-10 umwandeln und sezte Strings zusammen';

		IF fb_state_entry.E THEN
			Substring[1] := '';
			FOR i := 1 TO 10 BY 1 DO
				i_dint_to_hydra := st_data.iCounter[i];
				subr_Dint_to_Hydra_Counter();							(* Zähler in String umwandeln *)
				HelpString := CONCAT(sCounter, UINT_TO_STRING(i));
				HelpString := CONCAT(HelpString, '=');
				HelpString := CONCAT(HelpString, s_dint_to_hydra);
				HelpString := CONCAT(HelpString, sTrennzeichen);
				Substring[1] := CONCAT(Substring[1], HelpString);
			END_FOR
		END_IF

		(*-----------------------Weiterschaltbedingungen----------------------------*)
			fb_state_entry.i16_next_step:=142;
			
(*=======================================================*)
	142: fb_state_entry.s_debugtext:='Counter 10-20 umwandeln und sezte Strings zusammen';

		IF fb_state_entry.E THEN
			Substring[2] := '';
			FOR i := 11 TO 20 BY 1 DO
				i_dint_to_hydra := st_data.iCounter[i];
				subr_Dint_to_Hydra_Counter();							(* Zähler in String umwandeln *)
				HelpString := CONCAT(sCounter, UINT_TO_STRING(i));
				HelpString := CONCAT(HelpString, '=');
				HelpString := CONCAT(HelpString, s_dint_to_hydra);
				HelpString := CONCAT(HelpString, sTrennzeichen);
				Substring[2]:= CONCAT(Substring[2], HelpString);
			END_FOR
		END_IF

		(*-----------------------Weiterschaltbedingungen----------------------------*)
			fb_state_entry.i16_next_step:=144;
		
(*=======================================================*)
	144: fb_state_entry.s_debugtext:='Lese Daten und sezte Strings zusammen';

		IF fb_state_entry.E THEN
			(* Datum in das richtige Format bringen *)
			HelpString := MID(s_system_time, 2, 4);
			HelpString := CONCAT(HelpString, '/');
			HelpString := CONCAT(HelpString, MID(s_system_time, 2, 1));
			HelpString := CONCAT(HelpString, '/');
			HelpString := CONCAT(HelpString, MID(s_system_time, 4, 7));
			sDatum := HelpString;

			(* Zeit in das richtige Format bringen *)
			sZeit := MID(s_system_time, 8, 12);

			(* Prüfe welcher Status aktiv ist. Der niedrigste Status wird in Datei eingetragen *)
			FOR i := 1 TO 999 BY 1 DO
				IF st_data.bStatus[i] THEN
					EXIT;	(* Verlasse Schleife *)
				END_IF
			END_FOR

			(* wenn kein Status aktiv ist, dann schreibe MSTAT@M100=    Ohne Zahl  *)
			(* Falls kein Produktionssignal, dann Nicht zugeordnet *)
			IF i < 999 THEN
				HelpString := CONCAT(sMSTAT, UINT_TO_STRING(i));
			ELSE
				HelpString := 'MSTAT=30000';
			END_IF

			Substring[3] := '';
			HelpString := CONCAT(HelpString, sTrennzeichen);
			HelpString := CONCAT(HelpString, sDatumPrefix);
			HelpString := CONCAT(HelpString, sDatum);
			HelpString := CONCAT(HelpString, sTrennzeichen);
			HelpString := CONCAT(HelpString, sZeitPrefix);
			HelpString := CONCAT(HelpString, sZeit);
			Substring[3] := HelpString;
		END_IF

		(*-----------------------Weiterschaltbedingungen----------------------------*)
		fb_state_entry.i16_next_step:=150;
		
(*=======================================================*)
	150: fb_state_entry.s_debugtext:='Datei erstellen';

		IF fb_state_entry.E THEN
		   	fbFileOpen.bExecute:=TRUE;
		END_IF

		(*-----------------------Weiterschaltbedingungen----------------------------*)
		IF fbFileOpen.bBusy THEN
			fb_state_entry.i16_next_step:=160;
		END_IF

(*=======================================================*)
	160: fb_state_entry.s_debugtext:='Datei erstellen';

		(*-----------------------Weiterschaltbedingungen----------------------------*)
		IF 	NOT fbFileOpen.bBusy THEN
			i:=1;						(*wichtig für Dateizusammenbau*)
			fbFileOpen.bExecute:=FALSE;
			IF 	fbFileOpen.bError THEN
				nErrIdOpen:=fbFileOpen.nErrId;
				fb_state_entry.i16_next_step:=200;
			ELSE
				hFile := fbFileOpen.hFile;	(* Sehr wichtig hFile für FilePuts und Fileclose übergeben *)
				fb_state_entry.i16_next_step:=170;
			END_IF
		END_IF

(*=======================================================*)
	170: fb_state_entry.s_debugtext:='String in Datei eintragen';

		IF fb_state_entry.E THEN
			fbFilePuts.sLine:=Substring[i];
			fbFilePuts.bExecute:=TRUE;
		END_IF

		(*-----------------------Weiterschaltbedingungen----------------------------*)
		IF  fbFilePuts.bBusy THEN
			fb_state_entry.i16_next_step:=180;
		END_IF

(*=======================================================*)
	180: fb_state_entry.s_debugtext:='String in Datei eintragen';

		(*-----------------------Weiterschaltbedingungen----------------------------*)
		IF 	NOT fbFilePuts.bBusy THEN
			fbFilePuts.bExecute:=FALSE;
			IF 	fbFilePuts.bError THEN
				nErrIdWrite:=fbFilePuts.nErrId;
				fb_state_entry.i16_next_step:=200;
			ELSE
				fb_state_entry.i16_next_step:=190;
			END_IF
		END_IF

(*=======================================================*)
	190: fb_state_entry.s_debugtext:='Schleife Substrings in Datei eintragen';

		IF fb_state_entry.E THEN
			i :=  i+1;
		END_IF

		(*-----------------------Weiterschaltbedingungen----------------------------*)
		IF i <= 3 THEN
			fb_state_entry.i16_next_step:=170;
		ELSE
			fb_state_entry.i16_next_step:=200;
		END_IF

(*=======================================================*)
	200: fb_state_entry.s_debugtext:='Datei schließen';

		IF fb_state_entry.E THEN
			fbFileClose.bExecute:=TRUE;
		END_IF

		(*-----------------------Weiterschaltbedingungen----------------------------*)
		IF 	fbFileClose.bBusy THEN
			fb_state_entry.i16_next_step:=210;
		END_IF

(*=======================================================*)
	210: fb_state_entry.s_debugtext:='Datei schließen';

		(*-----------------------Weiterschaltbedingungen----------------------------*)
		IF NOT fbFileClose.bBusy THEN
			hFile := 0;
			fbFileClose.bExecute:=FALSE;
			IF 	fbFileClose.bError THEN
				nErrIdClose:=fbFileClose.nErrId;
				nErrIdCloseCounter := nErrIdCloseCounter + 1;
				fb_state_entry.i16_next_step:=FEHLER;
			ELSE
				fb_state_entry.i16_next_step:=300;
			END_IF
		END_IF

(*=======================================================*)
	300: fb_state_entry.s_debugtext:='Abfrage, kopiere Datei auf Server?';

		(*-----------------------Weiterschaltbedingungen----------------------------*)
		IF bKopiereDateiAufServer THEN
			fb_state_entry.i16_next_step:=310;
		ELSE
			Busy := FALSE;
			Done := TRUE;
			fb_state_entry.i16_next_step:=BEREIT;
		END_IF

(*=======================================================*)
	310: fb_state_entry.s_debugtext:='Kopiere Datei auf Server';

		IF fb_state_entry.E THEN
			DateiAufServerSpeichern.START := TRUE;
		END_IF

		(*-----------------------Weiterschaltbedingungen----------------------------*)
		IF DateiAufServerSpeichern.BUSY THEN
			fb_state_entry.i16_next_step:=320;
		ELSIF fb_state_entry.fb_ton_Step.ET >= T#2s THEN
			fb_state_entry.i16_next_step:=FEHLER;
		END_IF

		IF fb_state_entry.X THEN
			DateiAufServerSpeichern.START := FALSE;
		END_IF

(*=======================================================*)
	320: fb_state_entry.s_debugtext:='Warte bis fertig';

		(*-----------------------Weiterschaltbedingungen----------------------------*)
		IF NOT DateiAufServerSpeichern.BUSY AND
			NOT DateiAufServerSpeichern.ERR THEN
			fb_state_entry.i16_next_step:=330;
		ELSIF fb_state_entry.fb_ton_Step.ET >= T#5s THEN
			fb_state_entry.i16_next_step:=FEHLER;
		END_IF

(*=======================================================*)
	330: fb_state_entry.s_debugtext:='fertig';

		(*-----------------------Weiterschaltbedingungen----------------------------*)
		Busy := FALSE;
		Done := TRUE;
		fb_state_entry.i16_next_step:=BEREIT;

(*=======================================================*)
	FEHLER:
		IF fb_state_entry.E THEN
			Error := TRUE;
		END_IF

		(*-----------------------Weiterschaltbedingungen----------------------------*)
		fb_state_entry.i16_next_step:=BEREIT;

END_CASE


fb_state_entry(i16_pos:= 2);



fbFindFiles(
	bExecute	:= ,
	sNetId		:= '',
	sPathName	:= sFileName,
	pFindList	:= ADR(fbFindFilesEntry),
	cbFindList	:= SIZEOF(fbFindFilesEntry),
	tTimeout	:= t#15s );

 fbFileOpen(
	sNetId:='',
	sPathName:= sFileName,
	nMode:=FOPEN_MODEAPPEND,
	ePath:=PATH_GENERIC,
	bExecute:= ,
	tTimeout:=T#15s,
	hFile=> );

fbFilePuts(
	sNetId:='',
	hFile:=hFile,
	sLine:= ,
	bExecute:= ,
	tTimeout:=t#15s);

fbFileClose(
	sNetId:='',
	hFile:=hFile,
	bExecute:= ,
	tTimeout:=t#15s);

DateiAufServerSpeichern(
	NETID:='',
	PATHSTR	:='C:\Windows\System32\wscript.exe',
	DIRNAME	:=sPathStrDateiAufServerSpeichern,
	COMNDLINE	:='HydraDateiAufServerSpeichern.vbs',
	START		:=,
	TMOUT		:=T#10s);
END_FUNCTION_BLOCK
ACTION subr_Dint_to_Hydra_Counter:
(* Damit nur noch 4 Stellen übrig bleiben *)
i_dint_to_hydra := i_dint_to_hydra MOD 10000;

s_dint_to_hydra := DINT_TO_STRING(i_dint_to_hydra);
(* vordere Stellen mit 0 auffüllen *)
WHILE(LEN(s_dint_to_hydra) < 4) DO
	s_dint_to_hydra := CONCAT('0', s_dint_to_hydra);
END_WHILE
END_ACTION

(* POU zLibrary/Keyence/FB_KeyenceEtherCat, ST *)
FUNCTION_BLOCK FB_KeyenceEtherCat
VAR_INPUT
	st_ctrl_in						: struct_ctrl_in;
	JobNo							: INT;
	sConfig							: st_config_Keyence;	(*Initialisierung der Kamera*)
END_VAR
VAR_OUTPUT
	st_ctrl_out						: struct_ctrl_out;
	Connected						: BOOL;
	ActJobNo						: INT;
	b_Kam_Pruef_IO				: BOOL; 				(* Kameraprüfung Ergebnis iO *)
	b_Kam_Pruef_NIO				: BOOL; 				(* Kameraprüfung Ergebnis niO *)
	RecvDataString					: T_MaxString;
END_VAR
VAR
	b_Test							: BOOL;

	fb_ton_quitt						: TON;
	fb_state_entry					: ST_StateEntry;

 	BtnConnect						: sButtonVisu;
	BtnTrigger						: sButtonVisu;

	sm_kamera_keine_reaktion		: BOOL := FALSE;
	sm_kamera_nicht_bb			: BOOL := FALSE;
	sm_jobnummer_nicht_erlaubt		: BOOL := FALSE;		(* erlaubter Bereich von 0-15 *)
	sm_kamera_controler_error		: BOOL := FALSE;

	i								: INT;
	nInByte							: BYTE;

	stControl						: st_ctrl_out_Keyence;

	FB_ReadXmlLineConf			: FB_ReadXmlLine;
	FB_ReadXmlLineMsg			: FB_ReadXmlLine;
	(*Variablen für Behr Meldungen*)
	TempErrorText					: STRING(255);
	ProcessTime					: DINT;				(* Counts the time in steps of 100ms since starting operation *)
	Error							: ErrorStruct;

(*DL-EC1A: PDO-Kommunikation (Prozessdaten-Objekte)*)

	(*Input Request*)
	anInputRequest					AT%Q* 	: ARRAY [0..4] OF DWORD;

	(*Status of System*)
	bError_Status_00				AT%I*	: BOOL;		(* *)
(*	nError_Code_00					AT%I*	: UINT;							*)

	(*ID Current Value*)
(*	anTool_Score					AT%I* 	: ARRAY [0..7] OF DINT;			*)

	(*ID Status*)
	bChange_Program_Ack 			AT%I*	: BOOL;							
	bChange_Program_Failed			AT%I*	: BOOL;							
(*	bResult_Valid_00				AT%I*	: BOOL;
	bTotal_Status_OK_00				AT%I*	: BOOL;

	bResult_Valid_01				AT%I*	: BOOL;
	bRegist_Master_Image_Ack		AT%I*	: BOOL;
	bRegist_Master_Image_Failed		AT%I*	: BOOL;							*)
	bTotal_Status_OK_01				AT%I*	: BOOL;
	bTotal_Status_NG				AT%I*	: BOOL;
(*	bError_status					AT%I*	: BOOL;
	bClear_Error_Ack				AT%I*	: BOOL;							*)
	bRun							AT%I*	: BOOL;
	bBusy							AT%I*	: BOOL;
	bTrigger_Ready					AT%I*	: BOOL;
	bTrigger_Ack					AT%I*	: BOOL;
(*	bTrigger_Failed					AT%I*	: BOOL;
	bResult_Updated_Toggle			AT%I*	: BOOL;
	bCount_Up_Ack					AT%I*	: BOOL;
	bReset_Statistics_Ack			AT%I*	: BOOL;
	bReset_Count_Ack				AT%I*	: BOOL;

	abTool_Invalid					AT%I* 	: ARRAY [0..6] OF BOOL;
	abTool_State					AT%I* 	: ARRAY [0..6] OF BOOL;			*)
	abProgram_Num					AT%I* 	: ARRAY [0..6] OF BOOL;			
(*	abLogic							AT%I* 	: ARRAY [0..4] OF BOOL;

	bSD_Card_Detected				AT%I*	: BOOL;
	bSD_Save_Stop_Ack				AT%I*	: BOOL;
	bSD_Card_No_Space				AT%I*	: BOOL;

	(*WcState*)
	bWcState						AT%I*	: BOOL;
	bInputToggle					AT%I*	: BOOL;							*)

	(*Info Data*)
	nState							AT%I*	: UINT;
(*	bAdsAddr						AT%I*	: ARRAY [0..5] OF USINT;		*)

END_VAR
(* Zeiten *)
fb_ton_quitt(IN:= , PT:= t#100ms, Q=> , ET=> );

(* Aufrufe *)
	Btn_Init();
	Control();
	ErrorHandling();

(* Toplevel *)
IF	sConfig.Aktiv THEN
	IF 	NOT Connected THEN
		sm_kamera_nicht_bb := TRUE;
		fb_state_entry.i16_next_step := FEHLER;
	END_IF
ELSE
	fb_state_entry.i16_next_step := INAKTIV;
END_IF

IF fb_state_entry.i16_next_step > INIT AND fb_state_entry.i16_next_step < FEHLER THEN
	IF fb_state_entry.i16_next_step < STOP THEN
		IF 	st_ctrl_in.b_stop THEN
			fb_state_entry.i16_next_step := STOP;
		END_IF
		IF 	bError_Status_00 THEN
			sm_kamera_controler_error := TRUE;
			fb_state_entry.i16_next_step := FEHLER;
		END_IF
	END_IF
END_IF

(* ==================================Schrittkette================================ *)
fb_state_entry(i16_pos:= 1);

CASE fb_state_entry.i16_step OF
(*=======================================================*)
INIT_OBJ:
	fb_state_entry.i16_next_step := INIT;

(*=======================================================*)
INIT:
	IF 	fb_state_entry.E THEN
		fb_ton_quitt.IN := FALSE;
		st_ctrl_out := st_ctrl_out_Empty;

		b_Kam_Pruef_IO := FALSE;
		b_Kam_Pruef_NIO := FALSE;
		sm_kamera_nicht_bb := FALSE;
		sm_kamera_keine_reaktion := FALSE;
		sm_jobnummer_nicht_erlaubt := FALSE;
		sm_kamera_controler_error := FALSE;
		Error.No:=0;
		Error.Text:='';
	END_IF

	(*-----------------------Weiterschaltbedingungen----------------------------*)
	IF st_ctrl_in.b_init THEN
		fb_state_entry.i16_next_step := 20;
	END_IF

(*=======================================================*)
20: fb_state_entry.s_debugtext:='Reset';

	stControl.bReset:=TRUE;

	IF 	fb_state_entry.fb_ton_Step.ET > t#100ms THEN
		fb_state_entry.i16_next_step := BEREIT;
	END_IF

	IF 	fb_state_entry.X THEN
		stControl.bReset:=FALSE;
	END_IF

(*=======================================================*)
BEREIT: fb_state_entry.s_debugtext:='waiting for start';

	IF 	fb_state_entry.E THEN
		st_ctrl_out.b_bereit := TRUE;
	END_IF

	(*-----------------------Weiterschaltbedingungen----------------------------*)
	IF	st_ctrl_in.b_start THEN
		b_Kam_Pruef_IO := FALSE;
		b_Kam_Pruef_NIO := FALSE;
		fb_state_entry.i16_next_step := 110;
	END_IF

	IF 	fb_state_entry.X THEN
		st_ctrl_out.b_busy := TRUE;
		st_ctrl_out.b_bereit := FALSE;
		st_ctrl_out.b_fertig := FALSE;
	END_IF

(*=======================================================*)
110: fb_state_entry.s_debugtext:='check job number';

	IF 	fb_state_entry.E THEN
		stControl.bReset:=TRUE;
	END_IF

	(*-----------------------Weiterschaltbedingungen----------------------------*)

	IF 	JobNo <> ActJobNo THEN
		IF 	bRun AND
			NOT bBusy AND
			NOT bChange_Program_Ack THEN
				fb_state_entry.i16_next_step:=120;
		END_IF
	ELSE
		fb_state_entry.i16_next_step := 140;
	END_IF

	IF 	fb_state_entry.X THEN
		stControl.bReset:=FALSE;
	END_IF

(*=======================================================*)
120: fb_state_entry.s_debugtext:='set job number';

	IF 	fb_state_entry.E THEN
		IF 	JobNo < 0 AND JobNo > 15 THEN
			sm_jobnummer_nicht_erlaubt := TRUE;
			fb_state_entry.i16_next_step := FEHLER;
		ELSE
			stControl.bPrgChange:=TRUE;
			stControl.iJobNo:= JobNo;
		END_IF
	END_IF

	(*-----------------------Weiterschaltbedingungen----------------------------*)
	IF 	bChange_Program_Ack THEN
		fb_state_entry.i16_next_step:=130;
	ELSIF fb_state_entry.fb_ton_Step.ET > t#5s THEN
		sm_kamera_keine_reaktion := TRUE;
		fb_state_entry.i16_next_step := FEHLER;
	END_IF


	IF 	fb_state_entry.X THEN
		stControl.bPrgChange:=FALSE;
		stControl.iJobNo:= 0;
	END_IF

(*=======================================================*)
130: fb_state_entry.s_debugtext:='check job number';

	IF 	JobNo = ActJobNo AND
		NOT bChange_Program_Failed THEN
		fb_state_entry.i16_next_step := 140;
	END_IF

(*=======================================================*)
140: fb_state_entry.s_debugtext:='Reset and check Ready';

	IF 	fb_state_entry.E THEN
		stControl.bReset:=TRUE;
	END_IF

	(*-----------------------Weiterschaltbedingungen----------------------------*)

	IF 	bRun AND
		NOT bBusy AND
		bTrigger_Ready THEN
		fb_state_entry.i16_next_step:=150;
	END_IF

	IF 	fb_state_entry.X THEN
		stControl.bReset:=FALSE;
	END_IF

(*=======================================================*)
150: fb_state_entry.s_debugtext:='set trigger';

	stControl.bTrigger :=TRUE;
	(*-----------------------Weiterschaltbedingungen----------------------------*)
	IF 	bTrigger_Ack THEN
		fb_state_entry.i16_next_step:=160;
	ELSIF fb_state_entry.fb_ton_Step.ET > t#5s THEN
		sm_kamera_keine_reaktion := TRUE;
		fb_state_entry.i16_next_step := FEHLER;
	END_IF

	IF 	fb_state_entry.X THEN
		stControl.bTrigger:=FALSE;
	END_IF

(*=======================================================*)
160: fb_state_entry.s_debugtext:='result of camera';

	IF 	NOT bBusy AND
		bTotal_Status_OK_01 <> bTotal_Status_NG THEN
		b_Kam_Pruef_IO 	:= bTotal_Status_OK_01;
		b_Kam_Pruef_NIO := bTotal_Status_NG;
		fb_state_entry.i16_next_step := BEREIT;
	ELSIF fb_state_entry.fb_ton_Step.ET > t#5s THEN
		sm_kamera_keine_reaktion := TRUE;
		fb_state_entry.i16_next_step := FEHLER;
	END_IF

	IF 	fb_state_entry.X THEN
		st_ctrl_out.b_busy:=FALSE;
		st_ctrl_out.b_fertig := TRUE;
	END_IF

(*=======================================================*)
STOP, FEHLER:

	IF 	fb_state_entry.E THEN
		st_ctrl_out := st_ctrl_out_Empty;
		st_ctrl_out.b_gestoppt := fb_state_entry.i16_next_step = STOP;
		st_ctrl_out.b_fehler := fb_state_entry.i16_next_step = FEHLER;
		fb_ton_quitt.IN := FALSE;
	END_IF

		IF	sm_kamera_keine_reaktion THEN
			FB_ReadXmlLineMsg.ID:='sm_kamera_keine_reaktion';
			Error.No:=1;
		ELSIF
			sm_kamera_nicht_bb THEN
			FB_ReadXmlLineMsg.ID:='sm_kamera_nicht_bb';
			Error.No:=2;
		ELSIF
			sm_jobnummer_nicht_erlaubt THEN
			FB_ReadXmlLineMsg.ID:='sm_jobnummer_nicht_erlaubt';
			Error.No:=3;
		ELSIF
			sm_kamera_controler_error THEN
			FB_ReadXmlLineMsg.ID:='sm_kamera_controler_error';
			Error.No:=4;
		END_IF

	(*-----------------------Weiterschaltbedingungen----------------------------*)
	IF 	st_ctrl_in.b_quitt OR gResetAll THEN
		fb_ton_quitt.IN := TRUE;
	END_IF

	IF 	fb_ton_quitt.Q THEN
		fb_ton_quitt.IN := FALSE;
		fb_state_entry.i16_next_step := INIT;
	END_IF

(*=======================================================*)
INAKTIV:

	IF 	fb_state_entry.E THEN
		st_ctrl_out := st_ctrl_out_Empty;
	END_IF
	st_ctrl_out.b_bereit := TRUE;
	(*-----------------------Weiterschaltbedingungen----------------------------*)
	IF	sConfig.Aktiv THEN
		fb_state_entry.i16_next_step := INIT;
	END_IF

END_CASE

fb_state_entry(i16_pos:= 2);
st_ctrl_in := st_ctrl_in_Empty;
END_FUNCTION_BLOCK
ACTION Btn_Init:
(*=====================================================================*)
BtnConnect.Text:='Connect';
BtnConnect.BackgroundColor:=Color.darkgrey;
BtnConnect.Enable:= TRUE; (*ModeSelect.Mode <> MODE_MANUAL;*)
IF	BtnConnect.Enable THEN
	BtnConnect.TextColor:=Color.grey;
ELSE
	BtnConnect.TextColor:=Color.black;
END_IF
BtnConnect.Visible:=TRUE;

(*=====================================================================*)
BtnTrigger.Text:='Trigger';
BtnTrigger.BackgroundColor:=Color.darkgrey;
BtnTrigger.Enable:= TRUE; (* ModeSelect.Mode <> MODE_MANUAL;*)
IF	BtnTrigger.Enable THEN
	BtnTrigger.TextColor:=Color.grey;
ELSE
	BtnTrigger.TextColor:=Color.black;
END_IF
BtnTrigger.Visible:=TRUE;
END_ACTION
ACTION Control:
(* DL-EC1A: PDO-Kommunikation (Prozessdaten-Objekte)*)
			Connected:= nState = 8; 								(* 0x0008 = Slave in 'OP' state *)

(* Index: 7000  SubIndex: 1 - 5 *)

FOR i := 0 TO 4 DO
(*Bit 0*) 	anInputRequest[i].0:=stControl.bReset;					(*Reserviert (alles zurücksetzen)*)
END_FOR

(*Bit 1*) 	anInputRequest[0].1:=stControl.bPrgChange;				(*Programmwechselanforderung*)
			anInputRequest[1].1:=stControl.iJobNo.0;
			anInputRequest[2].1:=stControl.iJobNo.1;
			anInputRequest[3].1:=stControl.iJobNo.2;
			anInputRequest[4].1:=stControl.iJobNo.3;

			ActJobNo.0:=abProgram_Num[0];
			ActJobNo.1:=abProgram_Num[1];
			ActJobNo.2:=abProgram_Num[2];
			ActJobNo.3:=abProgram_Num[3];

(*Bit 2*) 	anInputRequest[0].2:=stControl.bTrigger;				(*Trigger*)

(*nicht benutzt*)
(*Bit 3*) 	anInputRequest[0].3	:=stControl.bMaster;				(*Master-Registrierunganforderung *)
(*Bit 4*) 	anInputRequest[0].4	:=stControl.bSpeicherstopp;			(*Speicherstopp SD-Karte Anfrage*)
(*Bit 5*) 	anInputRequest[0].5	:=stControl.bStatistikruecksetzung;	(* Statistikrücksetzung anfordern*)
(*Bit 6*) 	anInputRequest[0].6	:=stControl.bFehlerLoeschen;		(*Anforderung Fehler löschen*)
(*Bit 7*) 	anInputRequest[0].7	:=stControl.OCR_Seriennummer;		(*Anforderung OCR-Seriennummer Hochzählen*)
(*Bit 8*) 	anInputRequest[0].8	:=stControl.Zaehlung_Ruecksetzen;	(*Zählung-Rücksetzen Anforderung*)
(*Bit 9*) 	anInputRequest[0].9	:=stControl.Statistik_Ruecksetzen;	(*Anforderung Statistik aller Programme Rücksetzen*)
(*Bit 10*) 	anInputRequest[0].10:=stControl.Reserviert_10;
(*Bit 11*) 	anInputRequest[0].11:=stControl.Reserviert_11;
(*Bit 12*) 	anInputRequest[0].12:=stControl.Reserviert_12;
(*Bit 13*) 	anInputRequest[0].13:=stControl.Reserviert_13;
(*Bit 14*) 	anInputRequest[0].14:=stControl.Reserviert_14;
(*Bit 15*) 	anInputRequest[0].15:=stControl.Reserviert_15;
END_ACTION
ACTION ErrorHandling:
(*------------------------------------------------------------------
	Error-Handling
  ------------------------------------------------------------------*)

FB_ReadXmlLineConf(
	Prefix:= 'CONFIG',
	ID:= sConfig.InstName,
	File:= 'CONFIG.xml',
	Text=>  );

FB_ReadXmlLineMsg(
	Prefix:= 'MSG',
	ID:= ,
	File:= 'MSG.xml',
	Text=>);

IF	NOT st_ctrl_out.b_fehler OR NOT sConfig.Aktiv THEN
	Error.No:=0;
	Error.Text:='';
	TempErrorText:='';
END_IF

IF 	Error.Text<>''	AND ST_Lng.b_EndChangeLng THEN
	Error.Typ:=0;
	ErrorHandler.AddError(ErrorToAdd:=Error,
						sVisu:=Visu.ErrorHandler);
END_IF

IF	 st_ctrl_out.b_fehler THEN
	Error.Text:=FB_ReadXmlLineConf.Text;
	Error.Text:=CONCAT(Error.Text,': ');
	Error.Text:=CONCAT(Error.Text,FB_ReadXmlLineMsg.Text);
END_IF
END_ACTION

(* POU Stations/ST_02_RT_Tampondrucker/ST02_FBs/FB_Schwenken, ST *)
FUNCTION_BLOCK FB_Schwenken
VAR_INPUT
	b_quitt						: BOOL;
	b_0_grad					: BOOL;
	b_180_grad					: BOOL;
	b_90_grad					: BOOL;

END_VAR
VAR_IN_OUT
	ST02_90_180					: FB_Valve; 			(* 90 - 180 Grad (Valve) *)
	ST02_90_0					: FB_Valve; 			(* 90 - 0 Grad (Valve) *)
	ST02_90						:FB_ValveSensor;		 (* Schwenkarm 1 90 Grad*)
END_VAR

VAR_OUTPUT

	b_ready						: BOOL;
	b_done						: BOOL;
	b_busy						: BOOL;
	b_error						: BOOL;

	ST02_90_0_sens				: BOOL; 		(* 90 - 0 Grad (Sensor) *)
	ST02_90_sens				: BOOL;		(* 90 Grad (Sensor)*)
	ST02_90_180_sens			: BOOL; 		(* 90 - 180 Grad (Sensor) *)

END_VAR
VAR
	b_first_cycle						: BOOL := TRUE;
	fb_ton_wz						: TON;
	fb_ton_uez						: TON;
	fb_ton_quitt						: TON;
	fb_state_entry						: ST_StateEntry;
	fb_r_trig_start						: R_TRIG;
	fb_r_trig_init						: R_TRIG;
END_VAR

VAR_OUTPUT

END_VAR
VAR

END_VAR
IF b_first_cycle THEN
	b_first_cycle := FALSE;
END_IF

(* Zeiten *)
fb_ton_wz(IN:= , PT:= , Q=>  , ET=> );
fb_ton_uez(IN:= , PT:=DINT_TO_TIME(ST02_90_180.sInit.MaxTime * 4)  , Q=>  , ET=> );
fb_ton_quitt(IN:= , PT:= t#100ms, Q=> , ET=> );

ST02_90_0_sens:=ST02_90_0.SensorWorkIn[1].SensorSignal ; 				(* 90 - 0 Grad (Sensor) *)
ST02_90_sens:=ST02_90.ValveSensor;									(* 90 Grad (Sensor) *)
ST02_90_180_sens:=ST02_90_180.SensorWorkIn[1].SensorSignal; ; 			(* 90 - 180 Grad (Sensor) *)

(* Flanken *)
fb_r_trig_start(CLK:= b_0_grad OR b_90_grad OR b_180_grad, Q=> );

b_error := ST02_90_0.State < 0 OR ST02_90_180.State < 0;

IF	b_error THEN
	fb_state_entry.i16_next_step := FEHLER;
END_IF

fb_r_trig_init(CLK:=ModeSelect.Mode<=MODE_MANUAL);
IF	fb_r_trig_init.Q THEN
	fb_state_entry.i16_next_step := INIT;
END_IF

(* ==================================Schrittkette================================ *)
fb_state_entry(i16_pos:= 1, );

CASE fb_state_entry.i16_step OF
(*=======================================================*)
	INIT_OBJ:
		fb_state_entry.i16_next_step := INIT;


(*=======================================================*)
	INIT:
		IF fb_state_entry.E THEN
			fb_ton_wz.IN := FALSE;
			fb_ton_uez.IN := FALSE;
			b_ready := FALSE;
			b_done := FALSE;
			b_busy := FALSE;
			b_0_grad := FALSE;
			b_90_grad := FALSE;
			b_180_grad := FALSE;
		END_IF

		(*-----------------------Weiterschaltbedingungen----------------------------*)
		fb_state_entry.i16_next_step := BEREIT;

(*=======================================================*)
	BEREIT:
		IF fb_state_entry.E THEN
			b_ready := TRUE;
		END_IF

		(*-----------------------Weiterschaltbedingungen----------------------------*)
			IF 	fb_r_trig_start.Q  AND NOT b_error THEN
				IF	b_0_grad THEN
					fb_state_entry.i16_next_step := 110;
				ELSIF b_90_grad THEN
					fb_state_entry.i16_next_step := 200;
				ELSIF b_180_grad THEN
					fb_state_entry.i16_next_step := 300;
				END_IF
			END_IF

		IF fb_state_entry.X THEN
			b_busy := TRUE;
			b_done := FALSE;
			b_0_grad := FALSE;
			b_90_grad := FALSE;
			b_180_grad := FALSE;
			fb_ton_uez.IN:=FALSE;
		END_IF

(*=======================================================*)
	110:(*auf 0 Grad*)

		ST02_90_180.MoveInit:=TRUE;		(*Schwenkarm 1 drehen 90 - 180 Grad (Valve) *)
		ST02_90_0.MoveWork:=TRUE;	 	(*Schwenkarm 1 drehen 90 - 0 Grad (Valve) *)
		fb_state_entry.i16_next_step := 120;

	120:
		IF 	fb_state_entry.E THEN
			fb_ton_uez.IN:=TRUE;
		END_IF

		(*-----------------------Weiterschaltbedingungen----------------------------*)
		IF 	(ST02_90_180.State =STATE_OK AND
			ST02_90_0.State =STATE_OK) OR
			ST02_90_0.SensorWorkIn[1].SensorSignal   THEN
			b_done := TRUE;
			b_busy := FALSE;
			fb_state_entry.i16_next_step := BEREIT;
		END_IF

		IF	fb_ton_uez.Q THEN
			fb_state_entry.i16_next_step := FEHLER;
		END_IF

		IF fb_state_entry.X THEN
			fb_ton_uez.IN:=FALSE;
		END_IF

(*=======================================================*)
	200:(*auf 90 Grad*)

		ST02_90_180.MoveInit:=TRUE;		(*Schwenkarm 1 drehen 90 - 180 Grad (Valve) *)
		ST02_90_0.MoveInit:=TRUE;	 		(*Schwenkarm 1 drehen 90 - 0 Grad (Valve) *)
		fb_state_entry.i16_next_step := 210;

	210:
		IF 	fb_state_entry.E THEN
			fb_ton_uez.IN:=TRUE;
		END_IF

		(*-----------------------Weiterschaltbedingungen----------------------------*)
		IF 	(ST02_90_180.State =STATE_OK AND
			ST02_90_0.State =STATE_OK) OR
			ST02_90.ValveSensor THEN
			b_done := TRUE;
			b_busy := FALSE;
			fb_state_entry.i16_next_step := BEREIT;
		END_IF

		IF	fb_ton_uez.Q THEN
			fb_state_entry.i16_next_step := FEHLER;
		END_IF

		IF fb_state_entry.X THEN
			fb_ton_uez.IN:=FALSE;
		END_IF

(*=======================================================*)
	300:(*auf 0 Grad*)

		ST02_90_180.MoveWork:=TRUE;		(*Schwenkarm 1 drehen 90 - 180 Grad (Valve) *)
		ST02_90_0.MoveInit:=TRUE;	 		(*Schwenkarm 1 drehen 90 - 0 Grad (Valve) *)
		fb_state_entry.i16_next_step := 310;

	310:
		IF 	fb_state_entry.E THEN
			fb_ton_uez.IN:=TRUE;
		END_IF

		(*-----------------------Weiterschaltbedingungen----------------------------*)
		IF 	(ST02_90_180.State =STATE_OK AND
			ST02_90_0.State =STATE_OK) OR
			ST02_90_180.SensorWorkIn[1].SensorSignal   THEN
			b_done := TRUE;
			b_busy := FALSE;
			fb_state_entry.i16_next_step := BEREIT;
		END_IF

		IF	fb_ton_uez.Q THEN
			fb_state_entry.i16_next_step := FEHLER;
		END_IF

		IF fb_state_entry.X THEN
			fb_ton_uez.IN:=FALSE;
		END_IF
(*=======================================================*)
	FEHLER:
		IF fb_state_entry.E THEN
			b_error := TRUE;
			fb_ton_quitt.IN := FALSE;
		END_IF

		(*-----------------------Weiterschaltbedingungen----------------------------*)
		IF  NOT fb_state_entry.E AND NOT b_error THEN
			fb_ton_quitt.IN := TRUE;
		END_IF

		IF fb_ton_quitt.Q THEN
			fb_ton_quitt.IN := FALSE;
			fb_state_entry.i16_next_step := INIT;
		END_IF

(*=======================================================*)
	STOP:
		IF fb_state_entry.E THEN
			fb_ton_quitt.IN := FALSE;
		END_IF

		(*-----------------------Weiterschaltbedingungen----------------------------*)
		IF b_quitt AND NOT fb_state_entry.E THEN
			fb_ton_quitt.IN := TRUE;
		END_IF

		IF fb_ton_quitt.Q THEN
			fb_ton_quitt.IN := FALSE;
			fb_state_entry.i16_next_step := INIT;
		END_IF

END_CASE

fb_state_entry(i16_pos:= 2 );
END_FUNCTION_BLOCK

(* POU zLibrary/Valve/FB_Valve, ST *)
FUNCTION_BLOCK FB_Valve (*01.DEZ 2010,  B.Happach*)
VAR_OUTPUT
	State					: StateObject;		(* State of the object *)
	HomePosition			: BOOL;				(* object in home-position*)
	InitPosition				: BOOL;				(* Reflectet SensorState - All sensors showing "Init" *)
	WorkPosition			: BOOL;				(* Reflectet SensorState - All sensors showing "Work" *)
	ValveWorkOut			: ARRAY[1..8] OF sValveSensor_ValveOut; (* Structure To Sensorobject - Index is set in Init from Sensor *)
	ValveInitOut				: ARRAY[1..8] OF sValveSensor_ValveOut; (* Structure To Sensorobject - Index is set in Init from Sensor *)

END_VAR
VAR_INPUT
	MoveWork				: BOOL; 			(* Move to Workposition *)
	MoveInit				: BOOL;				(* Move to Initposition *)
	Enable					: BOOL:=TRUE;		(* Enables the operations on the valve *)
	Reset					: BOOL; 			(* switch for resetting the object *)
	SFCCurrentStep			: STRING(80);		(* aktually step in the step flow chart *)
	SFCCurrentPOU			: STRING(80);		(* Name of the step flow chart *)
	sInit						: sValveInit;			(* Initializingvalues to the Instance *)
	strAnlayse				: STRING(255); 		(*String to analyse Lockings*)
	SensorWorkIn			: ARRAY[1..8] OF sValveSensor_SensorOut; (* States from Worksensors - Index is set in Init from Sensor *)
	SensorInitIn				: ARRAY[1..8] OF sValveSensor_SensorOut; (* States from Initsensors - Index is set in Init from Sensor *)
	fb_Ton_Reset			:TON;
	fb_rTrig_Reset			:R_TRIG;
	WorkPos				:BOOL;
	InitPos					:BOOL;
	i						:INT;
END_VAR
VAR_IN_OUT
	sVisu					: sValveVisu;   		(* Structure for Visualisation *)
END_VAR
VAR
	CoilA					AT %Q* : BOOL; 	(* For Moving to WorkPosition *)
	CoilB					AT %Q* : BOOL; 	(* For Moving to InitPosition *)
	CoilAState				: BOOL; 			(* State Of Coil A - Depending on Valvetype *)
	CoilBState				: BOOL; 			(* State Of Coil B - Depending on Valvetype *)

(* Init and Worksensor Handling *)
	NoOfWorkSensors			: DINT;			(* Counter of Worksensors - Incremented by Sensorobject while initialisation *)
	NoOfInitSensors				: DINT;			(* Counter of Initsensors - Incremented by Sensorobject while initialisation *)
	NoOfValveCoils				: DINT;			(* Number of ValveCoils - from Init Struct *)

	IdxWork					: DINT;			(* Index Variable use in For-Loops *)
	IdxInit						: DINT;			(* Index Variable use in For-Loops *)

	HiCountWork				: DINT;			(* Varibable To Cout Sensors wich are high *)
	LoCountWork				: DINT;			(* Varibable To Cout Sensors wich are low *)
	HiCountInit					: DINT;			(* Varibable To Cout Sensors wich are high *)
	LoCountInit					: DINT;			(* Varibable To Cout Sensors wich are low *)

	WorkSensors_AllHi			: BOOL;			(* Internal Used Flag  *)
	WorkSensors_AllLo			: BOOL;			(* Internal Used Flag  *)
	InitSensors_AllHi				: BOOL;			(* Internal Used Flag  *)
	InitSensors_AllLo			: BOOL;			(* Internal Used Flag  *)
(* Movement Handling *)
	WorkingStep				: DINT;			(* Index for StateMachine *)
	MoveWorkStored			: BOOL; 		(* Stored Command "Move to Workposition"  *)
	MoveInitStored				: BOOL;			(* Stored Command "Move to Initposition" *)

	DampBoth					: BOOL;			(* This flag is Set when Damp both is required and possible *)
	DampBothTimer				: TON;			(* This Timer is used to set both valvecoils to fill the zylinder from Both sides *)

	DfltTxtDescription			: STRING(80):='Not defined!';
	DfltTxtVisuWorkButtonText 	: STRING(80):='Work';
	DfltTxtVisuInitButtonText 	: STRING(80):='Init';

(* Init Handling *)
	InitStep						: INT;				(* Init Step StateMachine *)
	InstanceNo					: INT;				(* Instance No for Language Handling - Used for Global Class functions *)
	InitState						: BOOL :=	FALSE;	(* Internal State for initialising *)

(* Visu Handling *)
	BtnMoveWork				: VisuButton;		(* Manage button *)
	BtnMoveInit					: VisuButton;		(* Manage button *)
	BtnReset					: VisuButton;		(* Manage button *)


(* Error Handling *)
	TimerTimeOut				: CheckProcTime;	(* Timer generates timeout signal *)
	ProcessTime				: DINT;				(* Counts the time since starting operation *)

	Error						: ErrorStruct;
	ErrorElapsed				: R_TRIG;

	LaufschriftErrh				: FB_Laufschrift;
	LaufschriftObj				: FB_Laufschrift_STR255;
	LaufschriftAnalyse			: FB_Laufschrift_STR255;
	TempString					: STRING(255);

	FB_ReadXmlLineConf		: FB_ReadXmlLine;
	FB_ReadXmlLineMsg		 : FB_ReadXmlLine;

END_VAR


(*Description kind of valve:
-------------------------------------
A	:	Valve with 1 coil  3/2 or 5/2 monostable
B	:	Valve with 2 coils 5/2 impulse
2G	:	Valve with 2 coils 2x 3/2
======================================*)

							
Error.No:=0;
Error.Text:='';

(*ermittel wo der Zylinder steht und schaltet das Ventil nach dem Reset auf die Position wo der Zylinder steht*)
WorkPos:=TRUE;
FOR i:=1 TO DINT_TO_INT(NoOfWorkSensors)  BY 1 DO
	IF	NOT SensorWorkIn[i].SensorSignal AND WorkPos THEN
		WorkPos:=FALSE;
	END_IF
END_FOR

InitPos:=TRUE;
FOR i:=1 TO DINT_TO_INT(NoOfInitSensors)  BY 1 DO
	IF	NOT SensorInitIn[i].SensorSignal AND InitPos THEN
		InitPos:=FALSE;
	END_IF
END_FOR
fb_Ton_Reset(IN:=NOT Reset, PT:=t#200ms);
fb_rTrig_Reset(CLK:=fb_Ton_Reset.Q);
IF	fb_rTrig_Reset.Q THEN
	MoveWork	:=WorkPos AND NoOfWorkSensors > 0; 			(* Move to Workposition *)
	MoveInit	:=InitPos AND NoOfInitSensors > 0; 				(* Move to Initposition *)
END_IF

(*------------------------------------------------------------------
	Initialization
  ------------------------------------------------------------------*)
IF 	NOT InitState THEN
	CASE InitStep OF

	0: (* Init Instance *)
			InitStep:=1;
	1: (* Init Internal OjbNo *)
			gValve.ObjCount:=gValve.ObjCount+1;
			InstanceNo:=gValve.ObjCount;
			InitStep:=50;

	50: (*Check KindOfValve*)
		IF 	sInit.KindOfValve='A' THEN
			NoOfValveCoils:=1;
			InitStep:=100;
		ELSIF
			sInit.KindOfValve='B' OR
			sInit.KindOfValve='2G' THEN
			NoOfValveCoils:=2;
			InitStep:=100;
		ELSE
			InitState:=FALSE;
			State:=STATE_ERROR;
			FB_ReadXmlLineMsg.ID:='KindOfValve';
			Error.No:=3;
			Error.Text:=sInit.InstName;
			Error.Text:=CONCAT(Error.Text,': ');
			Error.Text:=CONCAT(Error.Text,sInit.Description);
			Error.Text:=CONCAT(Error.Text,' - ');
			Error.Text:=CONCAT(Error.Text,FB_ReadXmlLineMsg.Text);
		END_IF

	100: (* Init Done *)
		InitState:=TRUE;
	END_CASE

END_IF (*InitState = FALSE*)

(* Add InitState to Global-Init-State to collect all Objects *)
gInitCollect:=gInitCollect AND InitState;

IF 	gInitOk THEN

	sVisu.Description			:= DfltTxtDescription;
	sVisu.WorkDescription		:= DfltTxtVisuWorkButtonText;
	sVisu.InitDescription			:= DfltTxtVisuInitButtonText;
(*------------------------------------------------------------------
	Show and Read Visu Buttons
  ------------------------------------------------------------------*)
	BtnMoveWork(Button:=sVisu.BtnMoveWork,
							Enable:= ModeSelect.Mode=MODE_MANUAL AND
									Enable AND
									(sInit.KindOfValve<>'2G' AND
									 NOT WorkPosition OR sInit.KindOfValve='2G' AND
									(NOT WorkPosition OR NOT CoilA)		) AND
									(State=STATE_WAIT OR State=STATE_ERROR),
							TextOn:=sVisu.WorkDescription
							);

	BtnMoveInit(Button:=sVisu.BtnMoveInit,
							Enable:=		ModeSelect.Mode=MODE_MANUAL AND
											Enable AND
											(	sInit.KindOfValve<>'2G' AND
												NOT InitPosition OR
												sInit.KindOfValve='2G' AND
											( 	NOT InitPosition OR NOT CoilB)		) AND
											(State=STATE_WAIT OR State=STATE_ERROR),
							TextOn:=sVisu.InitDescription
							);

	BtnReset(		Button:=sVisu.BtnReset,
							Enable:=ModeSelect.Mode=MODE_MANUAL ,
							TextOn:='Reset',
							);
END_IF

(*------------------------------------------------------------------
	Manual Mode
  ------------------------------------------------------------------*)
IF ModeSelect.Mode=MODE_MANUAL AND Enable THEN

	MoveWork:=MoveWork OR BtnMoveWork.Pressed;
	MoveInit:=MoveInit OR BtnMoveInit.Pressed;
	Reset:=Reset OR BtnReset.Pressed;
END_IF

(*------------------------------------------------------------------
	Sensor and Coil State Handling
  ------------------------------------------------------------------*)

(* Get States of All declarated Init Sensors *)
HiCountInit:=0;
LoCountInit:=0;
IF 	NoOfInitSensors>0 THEN
	FOR IdxInit:=1 TO NoOfInitSensors DO
		IF SensorInitIn[IdxInit].SensorSignal THEN
			HiCountInit:=HiCountInit+1;
		ELSE
			LoCountInit:=LoCountInit+1;
		END_IF
	END_FOR
END_IF
(* Get States of All declarated Work Sensors *)
HiCountWork:=0;
LoCountWork:=0;
IF 	NoOfWorkSensors>0 THEN
	FOR IdxWork:=1 TO NoOfWorkSensors DO
		IF SensorWorkIn[IdxWork].SensorSignal THEN
			HiCountWork:=HiCountWork+1;
		ELSE
			LoCountWork:=LoCountWork+1;
		END_IF
	END_FOR
END_IF

(* Handle Sensor States *)
InitSensors_AllHi:= (HiCountInit=NoOfInitSensors);
InitSensors_AllLo:= (LoCountInit=NoOfInitSensors);

WorkSensors_AllHi:= (HiCountWork=NoOfWorkSensors);
WorkSensors_AllLo:= (LoCountWork=NoOfWorkSensors);


(* Write Coilstates To Local Var - depending on Valvetype*)
IF 	NoOfValveCoils=1	THEN
	CoilAState:= CoilA;
	CoilBState:= NOT CoilA;
ELSE
		IF	sInit.KindOfValve='B' THEN
			IF 	NoOfWorkSensors>0 THEN
				CoilAState:=WorkSensors_AllHi AND InitSensors_AllLo ;
			ELSE
				CoilAState:=MoveWorkStored;
			END_IF

			IF 	NoOfInitSensors>0 THEN
				CoilBState:=InitSensors_AllHi AND WorkSensors_AllLo;
			ELSE
				CoilBState:=MoveInitStored;
			END_IF
		ELSE
			CoilAState:=CoilA AND NOT CoilB;
			CoilBState:=CoilB AND NOT CoilA;
		END_IF
END_IF

(* Handle Case if No Sensor Is declared *)
IF NoOfInitSensors>0 AND NoOfWorkSensors>0 THEN
	(* Work- and Initsensor available *)
	InitPosition:=InitSensors_AllHi AND WorkSensors_AllLo;
	WorkPosition:=WorkSensors_AllHi AND InitSensors_AllLo;
ELSIF
	NoOfInitSensors=0 AND NoOfWorkSensors>0 THEN
	(* Worksensor available and Initsensor NOT available *)
	WorkPosition:=WorkSensors_AllHi;
	InitPosition:=WorkSensors_AllLo AND CoilBState;
ELSIF
	NoOfInitSensors>0 AND NoOfWorkSensors=0 THEN
	(* Worksensor NOT available and Initsensor available *)
	InitPosition:=InitSensors_AllHi;
	WorkPosition:=InitSensors_AllLo AND CoilAState;
ELSIF
	NoOfInitSensors=0 AND NoOfWorkSensors=0 THEN
	(* If NO sensor is available then Inicate State over valvecoils*)
	InitPosition:=CoilBState;
	WorkPosition:=CoilAState;
END_IF

(*------------------------------------------------------------------
	Generate Damp Both Flag
  ------------------------------------------------------------------*)
DampBoth:=	sInit.KindOfValve='2G' AND
			sInit.DampBothTime>0 AND
			NOT (CoilA OR CoilB) AND
         			(   	MoveInit AND NOT InitPosition OR
             			MoveWork AND NOT WorkPosition );

(*------------------------------------------------------------------
	Move-Handling
  ------------------------------------------------------------------*)

CASE WorkingStep OF
	0: (* State STATE_WAIT *)

		IF	InitState THEN
			State:=STATE_WAIT;
			IF 	MoveWork OR
				MoveInit THEN
				WorkingStep:=100;
				TimerTimeOut.Start:=TRUE;
				State:=STATE_RUN;
				MoveWorkStored:=MoveWork;
				MoveInitStored:=MoveInit;
			END_IF
		END_IF

100:(* Move *)
		(* Check Damp Both *)
		IF DampBoth THEN
			WorkingStep:=110;
		ELSE
			WorkingStep:=120;
		END_IF
110:(* DampBoth *)
		DampBothTimer.IN:=TRUE;
		CoilA:=TRUE;
		CoilB:=TRUE;
		IF DampBothTimer.Q THEN
			WorkingStep:=120;
		END_IF
120: (* SET Valve Coils Move to Selected direction *)
		IF 	NoOfValveCoils=1 THEN
			CoilA:=MoveWorkStored;
			CoilB:=FALSE;
		ELSE
			CoilA:=MoveWorkStored;
			CoilB:=MoveInitStored;
		END_IF
		WorkingStep:=130;

130:(* Wait for Finishing movement *)
		IF 	(MoveWorkStored AND WorkPosition) OR
			(MoveInitStored AND InitPosition)	THEN
			WorkingStep:=140;
		END_IF
140:(* Reset Coils if necessary *)
		IF  sInit.KindOfValve='B' AND
			(	( NoOfWorkSensors>0 AND MoveWorkStored) OR
				( NoOfInitSensors>0 AND MoveInitStored) ) THEN
			CoilA:=FALSE;
			CoilB:=FALSE;
			WorkingStep:=1000;
		ELSE
			WorkingStep:=1000;
		END_IF
999: (* State Error *)
		State:=STATE_ERROR;
1000: (* State OK *)
		State:=STATE_OK;
		TimerTimeOut.Start:=FALSE;
		IF 	NOT MoveWork AND	NOT MoveInit OR
			MoveInit AND MoveWorkStored OR
			MoveWork AND MoveInitStored THEN
			WorkingStep:=0;
		END_IF
	END_CASE
	(*--------------------------------------------------------------------
		Handle Timeout
  --------------------------------------------------------------------*)
	IF TimerTimeOut.Timeout THEN
		State:=STATE_TIMEOUT;
		FB_ReadXmlLineMsg.ID:='timeout';
		Error.No:=1;
		Error.Text:=sInit.InstName;
		Error.Text:=CONCAT(Error.Text,': ');
		Error.Text:=CONCAT(Error.Text,sInit.Description);
		Error.Text:=CONCAT(Error.Text,' - ');
		Error.Text:=CONCAT(Error.Text,FB_ReadXmlLineMsg.Text);

		(* Set Flags to Raise Error in ValveSensor Object *)
		IF 	NoOfInitSensors>0 THEN
			FOR IdxInit:=1 TO NoOfInitSensors DO
				ValveInitOut[IdxInit].SignalHiExpected:=MoveInitStored;
				ValveInitOut[IdxInit].SignalLoExpected:=MoveWorkStored;
			END_FOR
		END_IF
		IF 	NoOfWorkSensors>0 THEN
			FOR IdxWork:=1 TO NoOfWorkSensors DO
				ValveWorkOut[IdxWork].SignalHiExpected:=MoveWorkStored;
				ValveWorkOut[IdxWork].SignalLoExpected:=MoveInitStored;
			END_FOR
		END_IF
	ELSE
		(* Reseet Flags to Raise Error in ValveSensor Object *)
		IF 	NoOfInitSensors>0 THEN
			FOR IdxInit:=1 TO NoOfInitSensors DO
				ValveInitOut[IdxInit].SignalHiExpected:=FALSE;
				ValveInitOut[IdxInit].SignalLoExpected:=FALSE;
			END_FOR
		END_IF
		IF 	NoOfWorkSensors>0 THEN
			FOR IdxWork:=1 TO NoOfWorkSensors DO
				ValveWorkOut[IdxWork].SignalHiExpected:=FALSE;
				ValveWorkOut[IdxWork].SignalLoExpected:=FALSE;
			END_FOR
		END_IF
	END_IF
	(*--------------------------------------------------------------------
		Handle unallowed Signalchange without Movecommand
  --------------------------------------------------------------------*)
	IF 	State=State_Wait AND
		NOT sInit.DisableSignalMonitoring THEN
		(* Set Flags to Raise Error in ValveSensor Object *)
		IF  	(MoveInitStored AND NOT InitPosition) OR
			(MoveWorkStored AND NOT WorkPosition)	THEN
			State:=STATE_ERROR;
			FB_ReadXmlLineMsg.ID:='SensorFault';
			Error.No:=1;
			Error.Text:=sInit.InstName;
			Error.Text:=CONCAT(Error.Text,': ');
			Error.Text:=CONCAT(Error.Text,sInit.Description);
			Error.Text:=CONCAT(Error.Text,' - ');
			Error.Text:=CONCAT(Error.Text, FB_ReadXmlLineMsg.Text);

			IF 	NoOfInitSensors>0 THEN
				FOR IdxInit:=1 TO NoOfInitSensors DO
					ValveInitOut[IdxInit].SignalHiExpected:=MoveInitStored;
					ValveInitOut[IdxInit].SignalLoExpected:=MoveWorkStored;
				END_FOR
			END_IF
			IF 	NoOfWorkSensors>0 THEN
				FOR IdxWork:=1 TO NoOfWorkSensors DO
					ValveWorkOut[IdxWork].SignalHiExpected:=MoveWorkStored;
					ValveWorkOut[IdxWork].SignalLoExpected:=MoveInitStored;
				END_FOR
			END_IF
		END_IF

	END_IF
	(*--------------------------------------------------------------------
		Call Timers
  --------------------------------------------------------------------*)
	TimerTimeOut(MTime:=sInit.MaxTime);
	DampBothTimer(PT:=DINT_TO_TIME(sInit.DampBothTime));
	(*--------------------------------------------------------------------
		Updating processtime (if State_RUN, STATE_TIMEOUT, STATE_RESETS, or STATE_STOPPED)
  --------------------------------------------------------------------*)
	IF	(State=State_RUN OR
		State=STATE_TIMEOUT OR
		State=STATE_RESETS OR
		State=STATE_STOPPED) AND
		sInit.MaxTime<>0 AND
		 ( NoOfInitSensors<>0 OR NoOfWorkSensors<>0)	THEN
		ProcessTime:=TimerTimeOut.PTime;
	END_IF
(*--------------------------------------------------------------------
	HomePosition
  --------------------------------------------------------------------*)

IF	sVisu.Description <> '' THEN
	CASE	sInit.HomePosDefine OF

	HOME_INIT:
		HomePosition:=InitPosition AND NOT WorkPosition AND (sInit.KindOfValve<>'2G' OR CoilBState);
	HOME_WORK:
		HomePosition:=WorkPosition AND NOT InitPosition AND (sInit.KindOfValve<>'2G' OR CoilAState);
	HOME_BOTH:
		HomePosition:=WorkPosition OR InitPosition;
	HOME_ALWAYS:
		HomePosition:=TRUE;
	ELSE
		HomePosition:=FALSE;
	END_CASE


(* Generating home position*)
	IF 	NOT HomePosition THEN
		ListHomeNOK(InstName:=sInit.InstName,Description:=FB_ReadXmlLineConf.Text);
	END_IF

	(* Object-homeposition concat with mainhomeposition *)
	gHomeOk:=gHomeOk AND HomePosition;
END_IF
(*------------------------------------------------------------------
	Update Visu
  ------------------------------------------------------------------*)
	sVisu.InstName:=sInit.InstName;

	sVisu.ProcessTime:=ProcessTime;
	sVisu.HomePosition:=HomePosition;
	sVisu.CoilA:=CoilA;
	sVisu.CoilB:=CoilB;
	sVisu.NoOfInitSensors:=NoOfInitSensors;
	sVisu.NoOfWorkSensors:=NoOfWorkSensors;
	sVisu.NoOfValveCoils:=NoOfValveCoils;

	sVisu.SAInitPosName:=SensorInitIn[1].SensorName;
	sVisu.SBInitPosName:=SensorInitIn[2].SensorName;
	sVisu.SCInitPosName:=SensorInitIn[3].SensorName;
	sVisu.SDInitPosName:=SensorInitIn[4].SensorName;
	sVisu.SEInitPosName:=SensorInitIn[5].SensorName;
	sVisu.SAWorkPosName:=SensorWorkIn[1].SensorName;
	sVisu.SBWorkPosName:=SensorWorkIn[2].SensorName;
	sVisu.SCWorkPosName:=SensorWorkIn[3].SensorName;
	sVisu.SDWorkPosName:=SensorWorkIn[4].SensorName;
	sVisu.SEWorkPosName:=SensorWorkIn[5].SensorName;

	sVisu.AInitPosition:=SensorInitIn[1].SensorSignal;
	sVisu.BInitPosition:=SensorInitIn[2].SensorSignal;
	sVisu.CInitPosition:=SensorInitIn[3].SensorSignal;
	sVisu.DInitPosition:=SensorInitIn[4].SensorSignal;
	sVisu.EInitPosition:=SensorInitIn[5].SensorSignal;
	sVisu.AWorkPosition:=SensorWorkIn[1].SensorSignal;
	sVisu.BWorkPosition:=SensorWorkIn[2].SensorSignal;
	sVisu.CWorkPosition:=SensorWorkIn[3].SensorSignal;
	sVisu.DWorkPosition:=SensorWorkIn[4].SensorSignal;
	sVisu.EWorkPosition:=SensorWorkIn[5].SensorSignal;

(*------------------------------------------------------------------
	Reset-Handling
  ------------------------------------------------------------------*)
IF 	Reset THEN
	State:=STATE_RESETS;
	WorkingStep:=0;
	ProcessTime:=0;
	TimerTimeOut.Start:=FALSE;
	DampBothTimer.IN:=FALSE;
	CoilA:=FALSE;
	CoilB:=FALSE;
	MoveWorkStored:=FALSE;
	MoveInitStored:=FALSE;
END_IF

(*------------------------------------------------------------------
	Error-Handling
  ------------------------------------------------------------------*)
ErrorElapsed(CLK:= Error.Text<>'');
IF ErrorElapsed.Q THEN
	Error.DateTime:=gVarDTSystemtime;
END_IF

IF Error.Text<>''	AND ST_Lng.b_EndChangeLng THEN
	Error.Typ:=0;
	(*Error.DateTime:=;*)
	ErrorHandler.AddError(
			ErrorToAdd:=Error,
			sVisu:=Visu.ErrorHandler);
END_IF

IF 	NOT Enable AND ModeSelect.Mode=MODE_MANUAL AND
	Error.Text='' AND strAnlayse<>''THEN

	strAnlayse:=CONCAT(' +++ gesperrt durch : ',strAnlayse);

	LaufschriftAnalyse(
	N:= 40,
	StepWidth:=1,
	PT:= t#100ms ,
	Text:= strAnlayse,
	Display=>sVisu.ErrorString );

	strAnlayse:='';
ELSE
	IF Error.Text<>'' THEN
		TempString:=CONCAT(' --- ',Error.Text);
		LaufschriftObj(
		N:= 40,
		StepWidth:=1,
		PT:= t#100ms ,
		Text:= TempString,
		Display=>sVisu.ErrorString );
	ELSE
		sVisu.ErrorString:='';
	END_IF
END_IF

(*------------------------------------------------------------------
	Reset Inputs
  ------------------------------------------------------------------*)
MoveWork		:=FALSE; 				(* Move to Workposition *)
MoveInit		:=FALSE;				(* Move to Initposition *)
Enable			:=FALSE; 				(* Enables the operations on the valve *)
Reset			:=FALSE; 				(* switch for resetting the object *)

sVisu.InstName:=sInit.InstName;
sVisu.BitName:=sInit.BitName;
sVisu.BtnMoveWork.Text:=sInit.WorkDescription;
sVisu.BtnMoveInit.Text:=sInit.InitDescription;
sVisu.ErrorPresent:=Error.Text<>'';

FB_ReadXmlLineConf(
	Prefix:= 'CONFIG',
	ID:= sInit.InstName,
	File:= 'CONFIG.xml',
	Text=> sVisu.Description );

FB_ReadXmlLineMsg(
	Prefix:= 'MSG',
	ID:= ,
	File:= 'MSG.xml',
	Text=>);


IF 	State = STATE_ERROR THEN
	Error.Text:=sInit.InstName;
	Error.Text:=CONCAT(Error.Text,': ');
	Error.Text:=CONCAT(Error.Text,sInit.Description);
	Error.Text:=CONCAT(Error.Text,' - ');
	Error.Text:=CONCAT(Error.Text,FB_ReadXmlLineMsg.Text);
END_IF
END_FUNCTION_BLOCK
ACTION AddInitSensor:
NoOfInitSensors:=NoOfInitSensors+1;
END_ACTION
ACTION AddWorkSensor:
NoOfWorkSensors:=NoOfWorkSensors+1;
END_ACTION

(* POU zLibrary/Valve/FB_ValveSensor, ST *)
FUNCTION_BLOCK FB_ValveSensor
VAR_INPUT
	ValveObject					: POINTER TO FB_Valve;		(* Pointer to declared Valve Instance *)
	sInit							: sValveSensorInit; 				(* Intialisation Informations e.g. Object Name *)
END_VAR
VAR_IN_OUT

END_VAR
VAR_OUTPUT
END_VAR
VAR
	ValveSensor	 			AT %I* :	BOOL; 					(* Sensor A InitPosition *)

	(* Sensor Handling *)
	ValveOut					: sValveSensor_ValveOut; 		(* Signals from Valve Object *)
	SensorOut					: sValveSensor_SensorOut;		(* Signals to Valve Object *)

	ValveSensorNo				: DINT; 							(* Number of Sensor given from ValveObject *)

	sVisuValveDummy			: sValveVisu; 					(* Dummy struct for Calling Action from Valve Object  *)

(* Init Handling *)
	InitState						: BOOL :=	FALSE;				(* Internal State for initialising *)
	InitStep						: INT;							(* Init Step StateMachine *)

(*  Error Handling *)
	Error						: ErrorStruct;						(* Local Error Struct *)
	ErrorElapsed				: R_TRIG;						(* Flag to Store Systemtime in Errorstruct when the error raising *)

	FB_ReadXmlLineConf		: FB_ReadXmlLine;
	FB_ReadXmlLineMsg		: FB_ReadXmlLine;
END_VAR
IF 	NOT InitState THEN
	CASE InitStep OF
	0: (* Init Instance *)
			InitStep:=100;

	100: (* Init Done *)

		IF	ValveSensorNo=0 THEN
			IF sInit.SensorType=sValveSensorType_INIT	THEN
		   		ValveObject^.AddInitSensor(sVisu:=sVisuValveDummy);
				ValveSensorNo:=ValveObject^.NoOfInitSensors;
			ELSE
		   		ValveObject^.AddWorkSensor(sVisu:=sVisuValveDummy);
				ValveSensorNo:=ValveObject^.NoOfWorkSensors;
			END_IF

			SensorOut.SensorName:=sInit.BitName;
			SensorOut.SensorType:=sInit.SensorType;

		END_IF

		InitState:=TRUE;
	END_CASE


ELSE
	(* Init State OK *)
	Error.No:=0;
	Error.Text:='';

	IF 	sInit.SensorType=sValveSensorType_INIT	THEN
		ValveOut:=ValveObject^.ValveInitOut[ValveSensorNo];
	ELSE
		ValveOut:=ValveObject^.ValveWorkOut[ValveSensorNo];
	END_IF

	(* Generate Errors  *)

	(* Check Signal Hi *)
	IF 	ValveOut.SignalHiExpected AND
		NOT ValveSensor	THEN
	  	Error.No:=1;
(*		Error.Text:=CONCAT(ValveObject^.sInit.InstName,' - ');*)
		FB_ReadXmlLineMsg.ID:='SensorFaultNotHigh';
		Error.Text:=CONCAT(Error.Text,sInit.InstName);
		Error.Text:=CONCAT(Error.Text,' :');
		Error.Text:=CONCAT(Error.Text,FB_ReadXmlLineConf.Text);
		Error.Text:=CONCAT(Error.Text,' - ');
		Error.Text:=CONCAT(Error.Text,FB_ReadXmlLineMsg.Text);

	END_IF


	(* Check Signal Low *)
	IF 	ValveOut.SignalLoExpected AND
		ValveSensor THEN
	  	Error.No:=1;
(*		Error.Text:=CONCAT(ValveObject^.sInit.InstName,' - ');*)
		FB_ReadXmlLineMsg.ID:='SensorFaultNotLow';
		Error.Text:=CONCAT(Error.Text,sInit.InstName);
		Error.Text:=CONCAT(Error.Text,' :');
		Error.Text:=CONCAT(Error.Text,FB_ReadXmlLineConf.Text);
		Error.Text:=CONCAT(Error.Text,' - ');
		Error.Text:=CONCAT(Error.Text,FB_ReadXmlLineMsg.Text);
	END_IF

	(* Write Sensor stete in local out Structure *)
	SensorOut.SensorSignal:=ValveSensor;

	(* Give local "out structure" to Valve object *)
	IF 	sInit.SensorType=sValveSensorType_INIT THEN
		ValveObject^.SensorInitIn[ValveSensorNo]:=SensorOut;
	ELSE
		ValveObject^.SensorWorkIn[ValveSensorNo]:=SensorOut;
	END_IF

END_IF

(*------------------------------------------------------------------
	Error-Handling
  ------------------------------------------------------------------*)

ErrorElapsed(CLK:= Error.Text<>'');
IF 	ErrorElapsed.Q THEN
	Error.DateTime:=gVarDTSystemtime;
END_IF

IF Error.Text<>''	AND ST_Lng.b_EndChangeLng THEN
	Error.Typ:=0;
	ErrorHandler.AddError(
				ErrorToAdd:=Error,
				sVisu:=Visu.ErrorHandler);
END_IF

(*------------------------------------------------------------------
	Language-Handling
  ------------------------------------------------------------------*)

FB_ReadXmlLineConf(
	Prefix:= 'CONFIG',
	ID:= sInit.InstName,
	File:= 'CONFIG.xml',
	Text=> );


